(* Logix 5000 project; controller Final vendor 1 type 14 code 242 rev 32.11; software revision 32.00 *)

TASK MainTask (continuous, watchdog 500 ms) : MainProgram
TASK SafetyTask (periodic, rate 20 ms, priority 10, watchdog 20 ms, safety) : SafetyProgram

MODULES
   Local : vendor 1 type 14 code 242 (5069 0, rev 32.11)
      IO_002 : 5069-IF8 (5069 2, rev 2.1, StandardDataDriven RPI 100 ms)
      IO_001 : 5069-IF8 (5069 1, rev 2.1, StandardDataDriven RPI 100 ms)
      IO_003 : 5069-IF8 (5069 3, rev 2.1, StandardDataDriven RPI 100 ms)
      IO_006 : vendor 1 type 7 code 394 (5069 6, rev 2.1, StandardDataDriven RPI 5 ms)
      IO_004 : vendor 1 type 7 code 395 (5069 4, rev 2.1, StandardDataDriven RPI 5 ms)
      IO_005 : vendor 1 type 7 code 395 (5069 5, rev 2.1, StandardDataDriven RPI 5 ms)
      IO_007 : vendor 1 type 109 code 90 (5069 7, rev 3.1, StandardDataDriven RPI 80 ms)
      EN_001 : 1734-AENTR (Ethernet 107.0.114.14, rev 5.1, Output RPI 20 ms)
         IO_008 : vendor 1 type 35 code 15 (PointIO 1, rev 2.1, Input RPI 10 ms, Output RPI 20 ms)
         IO_009 : vendor 1 type 35 code 16 (PointIO 2, rev 2.1, Input RPI 10 ms, Output RPI 20 ms)
END_MODULES

TYPE SensorType :   // To monitor the sensor readings, we use this data type
STRUCT
   CurrentValue : DINT;
   PreviousValue0 : DINT;
   PreviousValue1 : DINT;
   PreviousValue2 : DINT;
   PreviousValue3 : DINT;
   PreviousValue4 : DINT;
   PreviousValue5 : DINT;
   PreviousValue6 : DINT;
   PreviousValue7 : DINT;
   PreviousValue8 : DINT;
   PreviousValue9 : DINT;
   Mean10 : DINT;
   StanDev : DINT;
   State : DINT;
   Count : DINT;
   MeanStart : BOOL;
END_STRUCT
END_TYPE

VAR_GLOBAL   (* controller tags *)
   ACC_TIMER : DINT;
   AT : BOOL;
   B_NomCount : DINT;
   B_Pres0 : SensorType;   // Holds all values related to Brakes Pressure Sensor #0
   B_Pres1 : SensorType;   // Holds all values related to Brakes Pressure Sensor #1
   B_Pres2 : SensorType;   // Holds all values related to Brakes Pressure Sensor #2
   B_Pres3 : SensorType;   // Holds all values related to Brakes Pressure Sensor #3
   B_Pres4 : SensorType;   // Holds all values related to Brakes Pressure Sensor #4
   B_Pres5 : SensorType;   // Holds all values related to Brakes Pressure Sensor #5
   B_Pres6 : SensorType;   // Holds all values related to Brakes Pressure Sensor #6
   B_Pres7 : SensorType;   // Holds all values related to Brakes Pressure Sensor #7
   B_Pres8 : SensorType;   // Holds all values related to Brakes Pressure Sensor #8
   B_Pres9 : SensorType;   // Holds all values related to Brakes Pressure Sensor #9
   B_Tem0 : SensorType;   // Holds all values related to Brakes Temperature Sensor #0
   B_Tem1 : SensorType;   // Holds all values related to Brakes Temperature Sensor #1
   BAT_FLAG : DINT;
   BATTERY_CURRENT : DINT;
   BATTERY_TEMP : DINT;
   BATTERY_VOLTAGE : DINT;
   BRAKE_FLAG : DINT;
   BRAKE_SUBSTATE1 : DINT;
   BRAKE_SUBSTATE2 : DINT;
   C_Las0 : SensorType;   // Holds all values related to Controls Laser Sensor #0
   C_Las1 : SensorType;   // Holds all values related to Controls Laser Sensor #1
   CA : BOOL;
   CC : BOOL;
   CD1 : BOOL;
   CD2 : BOOL;
   CD3 : BOOL;
   COAST_TIMER : DINT;
   COAST_TONR : DINT;
   COMMAND : DINT;
   COMN_FLAG : DINT;
   CP1 : BOOL;
   CP2 : BOOL;
   CPX : BOOL;
   CT : BOOL;
   CurrentState : DINT;
   Initialized : DINT;
   P_NomCount : DINT;
   P_Pres0 : SensorType;   // Holds all values related to Pressure Pressure Sensor #0
   P_Pres1 : SensorType;   // Holds all values related to Pressure Pressure Sensor #1
   P_Pres2 : SensorType;   // Holds all values related to Pressure Pressure Sensor #2
   P_Pres3 : SensorType;
   P_Pres4 : SensorType;
   P_Tem0 : SensorType;   // Holds all values related to Pressure Temperature Sensor #0
   P_Tem1 : SensorType;   // Holds all values related to Pressure Temperature Sensor #1
   P_Tem2 : SensorType;
   P_Tem3 : SensorType;
   P_Tem4 : SensorType;
   POD_ACCELERATION : DINT;
   POD_DISTANCE : DINT;
   POD_TIME : DINT[2];
   POD_VELOCITY : DINT;
   PREV_ACCELERATION : DINT;
   PREV_DISTANCE : DINT;
   PREV_TIME : DINT[2];
   PREV_VELOCITY : DINT;
   PROP_FLAG : DINT;
   PROP_STATE : DINT;
   PROP_TNK_PRES : DINT;
   READY : BOOL;
   STATE : DINT;
   STRIPE_COUNT : DINT;
   SYSTEM_FAIL : DINT;
END_VAR

PROGRAM MainProgram   (* main routine MainRoutine *)
VAR
   ACC_TIMER : FBD_TIMER;
   COAST_TIMER : FBD_TIMER;
   SIMULATOR : FBD_TIMER;
END_VAR

ROUTINE A01_Initialize   (* structured text *)
// Initializes the values of all tags
   JSR(Initial_B_Pres0);
   JSR(Initial_B_Pres1);
   JSR(Initial_B_Pres2);
   JSR(Initial_B_Pres3);
   JSR(Initial_B_Pres4);
   JSR(Initial_B_Pres5);
   JSR(Initial_B_Pres6);
   JSR(Initial_B_Pres7);
   JSR(Initial_B_Pres8);
   JSR(Initial_B_Pres9);
   JSR(Initial_B_Tem0);
   JSR(Initial_B_Tem1);
   Local:5:O.Pt00.Data := 1;
   Local:5:O.Pt01.Data := 1;
   Local:5:O.Pt02.Data := 1;
   Local:5:O.Pt03.Data := 1;
   B_NomCount := 24; //Brakes Initialized
   JSR(Initial_C_Las0);
   JSR(Initial_C_Las1); //Controls Initialized
   JSR(Initial_P_Pres0);
   JSR(Initial_P_Pres1);
   JSR(Initial_P_Pres2);
   JSR(Initial_P_Pres3);
   JSR(Initial_P_Pres4);
   JSR(Initial_P_Tem0);
   JSR(Initial_P_Tem1);
   JSR(Initial_P_Tem2);
   JSR(Initial_P_Tem3);
   JSR(Initial_P_Tem4);
   Local:4:O.Pt00.Data := 1;
   Local:4:O.Pt01.Data := 0;
   Local:4:O.Pt02.Data := 0;
   Local:4:O.Pt03.Data := 1;
   P_NomCount := 20; //Propulsion Initialized
   BATTERY_CURRENT := 0;
   BATTERY_TEMP := 0;
   BATTERY_VOLTAGE := 0; //Power Initialized
   STRIPE_COUNT := 0;
   POD_DISTANCE := 0;
   POD_VELOCITY := 0;
   POD_ACCELERATION := 0;
   PREV_DISTANCE := 0;
   PREV_VELOCITY := 0;
   PREV_ACCELERATION := 0;
   READY := 0;
   //COAST_TIMER := 0;
   PROP_TNK_PRES := 0;
   PROP_STATE := 0;
   BRAKE_SUBSTATE1 := 0;
   BRAKE_SUBSTATE2 := 0;
   PROP_FLAG := 0;
   BRAKE_FLAG := 0;
   COMN_FLAG := 0;
   BAT_FLAG := 0;
   SYSTEM_FAIL := 0;
   STATE := 1;
   Initialized := 5380; //All Initialized
   //low-speed drive parameters missing
END_ROUTINE

ROUTINE A02_Update   (* structured text *)
// Updates all sensor value tags
   JSR(Update_B_Pres0);
   JSR(Update_B_Pres1);
   JSR(Update_B_Pres2);
   JSR(Update_B_Pres3);
   JSR(Update_B_Pres4);
   JSR(Update_B_Pres5);
   JSR(Update_B_Pres6);
   JSR(Update_B_Pres7);
   JSR(Update_B_Pres8);
   JSR(Update_B_Pres9);
   JSR(Update_B_Tem0);
   JSR(Update_B_Tem1); //Brakes Updated
   JSR(Update_C_Las0);
   JSR(Update_C_Las1); //Controls Updated
   JSR(Update_P_Pres0);
   JSR(Update_P_Pres1);
   JSR(Update_P_Pres2);
   JSR(Update_P_Pres3);
   JSR(Update_P_Pres4);
   JSR(Update_P_Tem0);
   JSR(Update_P_Tem1);
   JSR(Update_P_Tem2);
   JSR(Update_P_Tem3);
   JSR(Update_P_Tem4); //Propulsion Updated
   JSR(Update_Bat_Current);
   JSR(Update_Bat_Temp);
   JSR(Update_Bat_Voltage); //Power Updated
   JSR(Rx_Command);
   //limit switches
   //low-speed drive parameters
END_ROUTINE

ROUTINE A03_Process   (* structured text *)
// Processes input data
   //high speed counter interface
   STRIPE_COUNT := (C_Las0.CurrentValue + C_Las1.CurrentValue)/2; //2 can be substituted with nominal count of laser sensors
   
   PREV_DISTANCE := POD_DISTANCE;
   POD_DISTANCE := STRIPE_COUNT*3048; //units cm
   
   PREV_TIME[0] := POD_TIME[0];
   GSV(WallClockTime,,CurrentValue,POD_TIME[0]); //units microseconds
   
   PREV_VELOCITY := POD_VELOCITY;
   POD_VELOCITY := (POD_DISTANCE - PREV_DISTANCE)/(100000*(POD_TIME[0] - PREV_TIME[0])); //units cm/s
   
   PREV_ACCELERATION := POD_ACCELERATION;
   POD_ACCELERATION := (POD_VELOCITY - PREV_VELOCITY)/(POD_TIME[0] - PREV_TIME[0]); //units cm/s2
   
   //Process Data part 2
END_ROUTINE

ROUTINE A04_State   (* structured text *)
// Updates the state of the pod
   JSR(Check_Distance_1); //Checks if POD_DISTANCE >= 3000 cm
   JSR(Check_Distance_2); //Checks if POD_DISTANCE >= 80000 cm
   JSR(Check_Distance_3); //Checks if POD_DISTANCE >= 125000 cm
   JSR(Check_TankPres_1); //Checks if PROP_TNK_PRES >= 200 PSI
   JSR(Check_TankPres_2); //Checks if PROP_TNK_PRES <= 100 PSI
   JSR(Check_TankPres_X); //Checks if ACT_TNK_PRES == ??
   JSR(Check_PodAcc_1); //Checks if POD_ACCELERATION <= 0 cm/s2
   JSR(Check_AccTimer); // Checks if ACC_TIMER >= 7.7 sec
   JSR(Check_CoastTimer); //Checks if COAST_TIMER >= 10 sec
END_ROUTINE

ROUTINE A05_Actions   (* structured text *)
// Performs the state actions of the pod
   case STATE of
   	1: JSR(B01_Idle);
   	2: JSR(B02_SystemCheck);
   	3: JSR(B03_Armed);
   	4: JSR(B04_Acceleration);
   	5: JSR(B05_Coast);
   	6: JSR(B06_Brake);
   	7: JSR(B07_Stop);
   	8: JSR(B08_Crawl);
   	9: JSR(B09_End);
   	10: JSR(B10_EmergencyShutdown);
   end_case;
END_ROUTINE

ROUTINE A06_Relay   (* structured text *)
// Relays pod data to monitoring station
   //communication
END_ROUTINE

ROUTINE B01_Idle   (* structured text *)
   if COMMAND = 2 then
   	STATE := 2; //System Check
   end_if;
   
   if COMMAND = 9 then
   	STATE := 9; //End
   end_if;
   
   if COMMAND = 10 then
   	STATE := 10; //Emergency Shutdown
   end_if;
END_ROUTINE

ROUTINE B02_SystemCheck   (* structured text *)
   JSR(NomCheck_B1);
   JSR(NomCheck_P1);
   
   if B_NomCount <> 24 then
   	JSR(FaultTest_B);
   end_if;
   
   if P_NomCount <> 24 then
   	JSR(FaultTest_P);
   end_if;
   
   if COMMAND = 3 then
   	STATE := 3; //Armed
   end_if;
   
   if COMMAND = 1 then
   	STATE := 1; //Idle
   end_if;
   
   if COMMAND = 10 then
   	STATE := 10; //Emergency Shutdown
   end_if;
END_ROUTINE

ROUTINE B03_Armed   (* structured text *)
   if COMMAND = 4 then
   	STATE := 4; //Acceleration
   end_if;
   
   if COMMAND = 8 then
   	STATE := 8; //Crawl
   end_if;
   
   if COMMAND = 10 then
   	STATE := 10; //Emergency Shutdown
   end_if;
END_ROUTINE

ROUTINE B04_Acceleration   (* structured text *)
   ACC_TIMER.PRE := 10000;
   ACC_TIMER.TimerEnable := 1;
   ACC_TIMER.Reset := 0;
   TONR(ACC_TIMER);
   
   //EN_001:2:O.Pt01Data := 1;
   //EN_001:2:O.Pt02Data := 1;
   //EN_001:2:O.Pt00Data := 1; //Slow crawl
   
   if CD1 then //POD_DISTANCE >= 3000 cm?
   	//EN_001:2:O.Pt01Data := 0;
   	//EN_001:2:O.Pt02Data := 0;
   	//EN_001:2:O.Pt00Data := 0; //End crawl
   	READY := 1;
   end_if;
   //Timer to ready
   if READY then
   	Local:4:O.Pt01.Data := 1;
   	Local:4:O.Pt02.Data := 1; //Activate Propulsion
   end_if;
   
   if CPX then //TA-5 > 900 PSI?
   	Local:4:O.Pt00.Data := 0; //Special condition
   end_if;
   
   if CP1 AND CA then //PROP_TNK_PRES <= 200 PSI?
   	STATE := 5; //Coast
   end_if;
END_ROUTINE

ROUTINE B05_Coast   (* structured text *)
   COAST_TIMER.PRE := 7700;
   COAST_TIMER.TimerEnable := 1;
   COAST_TIMER.Reset := 0;
   TONR(COAST_TIMER); //Coast timer initialized
   
   Local:4:O.Pt01.Data := 0;
   Local:4:O.Pt02.Data := 0; //Propulsion disengaged
   
   if CP2 then
   	Local:4:O.Pt03.Data := 0; //Relief pressure valve open
   end_if;
   
   if CD2 OR CT OR (COMMAND = 7) then
   	STATE := 6; //Brake
   end_if;
   
   if COMMAND = 10 then
   	STATE := 10; //Emergency Shutdown
   end_if;
END_ROUTINE

ROUTINE B06_Brake   (* structured text *)
   Local:4:O.Pt03.Data := 1; //Relief pressure valve closed
   Local:5:O.Pt00.Data := 0;
   Local:5:O.Pt01.Data := 0;
   Local:5:O.Pt02.Data := 0;
   Local:5:O.Pt03.Data := 0; //Brakes engaged
   
   if POD_VELOCITY = 0 then
   	STATE := 7; //Stop
   end_if;
   
   if CA then
   	STATE := 10;
   end_if;
END_ROUTINE

ROUTINE B07_Stop   (* structured text *)
   Local:5:O.Pt00.Data := 1;
   Local:5:O.Pt01.Data := 1;
   Local:5:O.Pt02.Data := 1;
   Local:5:O.Pt03.Data := 1; //Disengage Brakes
   
   if COMMAND = 8 then
   STATE := 8; //Crawl
   end_if;
   
   if COMMAND = 9 then
   STATE := 9; //End
   end_if;
   
   if COMMAND = 10 then
   	STATE := 10; //Emergency Shutdown
   end_if;
END_ROUTINE

ROUTINE B08_Crawl   (* structured text *)
   //EN_001:2:O.Pt01Data := 1; // D = 1 Forward, D = 0 Backward
   //EN_001:2:O.Pt02Data := 1; //
   //EN_001:2:O.Pt00Data := 1; // pulse F at 4333 Hz //Slow crawl
   
   if CD3 OR (COMMAND = 7) then
   	//EN_001:2:O.Pt01Data := 0;
   	//EN_001:2:O.Pt02Data := 0;
   	//EN_001:2:O.Pt00Data := 0; //End crawl
   	STATE := 6; //Stop
   end_if;
END_ROUTINE

ROUTINE B09_End   (* structured text *)
   //Do nothing
END_ROUTINE

ROUTINE B10_EmergencyShutdown   (* structured text *)
   // Relay system faliure
   if CA then
   	Local:4:O.Pt01.Data := 0;
   	Local:4:O.Pt02.Data := 0; //Propulsion tanks closed
   end_if;
   Local:5:O.Pt00.Data := 0;
   Local:5:O.Pt01.Data := 0;
   Local:5:O.Pt02.Data := 0;
   Local:5:O.Pt03.Data := 0; //Brakes activated
   
   if CP2 then
   	STATE := 7; //Stop
   else
   	Local:4:O.Pt03.Data := 0; //Relief pressure valve
   	STATE := 7; //Stop
   end_if;
END_ROUTINE

ROUTINE Check_AccTimer   (* structured text *)
   if ACC_TIMER.DN then
   	AT := 1;
   	end_if;
END_ROUTINE

ROUTINE Check_CoastTimer   (* structured text *)
   if COAST_TIMER.DN then
   	CT := 1;
   	end_if;
END_ROUTINE

ROUTINE Check_Distance_1   (* structured text *)
   if POD_DISTANCE >= 3000 then
   	CD1 := 1;
   end_if;
END_ROUTINE

ROUTINE Check_Distance_2   (* structured text *)
   if POD_DISTANCE >= 80000 then
   	CD2 := 1;
   end_if;
END_ROUTINE

ROUTINE Check_Distance_3   (* structured text *)
   if POD_DISTANCE >= 125000 then
   	CD3 := 1;
   end_if;
END_ROUTINE

ROUTINE Check_LSDTimer   (* structured text *)
   
END_ROUTINE

ROUTINE Check_PodAcc_1   (* structured text *)
   if POD_ACCELERATION <= 0 then
   	CA := 1;
   end_if;
END_ROUTINE

ROUTINE Check_TankPres_1   (* structured text *)
   if (P_Pres1.CurrentValue + P_Pres2.CurrentValue + P_Pres3.CurrentValue + P_Pres4.CurrentValue) <= 200 then
   	CP1 := 1;
   end_if;
END_ROUTINE

ROUTINE Check_TankPres_2   (* structured text *)
   if (P_Pres1.CurrentValue + P_Pres2.CurrentValue + P_Pres3.CurrentValue + P_Pres4.CurrentValue) = 0 then
   	CP2 := 1;
   end_if;
END_ROUTINE

ROUTINE Check_TankPres_X   (* structured text *)
   if P_Pres0.CurrentValue < 250 then
   	CPX := 1;
   end_if;
END_ROUTINE

ROUTINE FaultTest_B   (* structured text *)
   
END_ROUTINE

ROUTINE FaultTest_P   (* structured text *)
   
END_ROUTINE

ROUTINE Initial_B_Pres0   (* structured text *)
   B_Pres0.CurrentValue := 0;
   B_Pres0.PreviousValue0 := 0;
   B_Pres0.PreviousValue1 := 0;
   B_Pres0.PreviousValue2 := 0;
   B_Pres0.PreviousValue3 := 0;
   B_Pres0.PreviousValue4 := 0;
   B_Pres0.PreviousValue5 := 0;
   B_Pres0.PreviousValue6 := 0;
   B_Pres0.PreviousValue7 := 0;
   B_Pres0.PreviousValue8 := 0;
   B_Pres0.PreviousValue9 := 0;
   B_Pres0.Count := 0;
   B_Pres0.Mean10 := 0;
   B_Pres0.StanDev := 0;
   B_Pres0.State := 0;
   B_Pres0.MeanStart := 0;
END_ROUTINE

ROUTINE Initial_B_Pres1   (* structured text *)
   B_Pres1.CurrentValue := 0;
   B_Pres1.PreviousValue0 := 0;
   B_Pres1.PreviousValue1 := 0;
   B_Pres1.PreviousValue2 := 0;
   B_Pres1.PreviousValue3 := 0;
   B_Pres1.PreviousValue4 := 0;
   B_Pres1.PreviousValue5 := 0;
   B_Pres1.PreviousValue6 := 0;
   B_Pres1.PreviousValue7 := 0;
   B_Pres1.PreviousValue8 := 0;
   B_Pres1.PreviousValue9 := 0;
   B_Pres1.Count := 0;
   B_Pres1.Mean10 := 0;
   B_Pres1.StanDev := 0;
   B_Pres1.State := 0;
   B_Pres1.MeanStart := 0;
END_ROUTINE

ROUTINE Initial_B_Pres2   (* structured text *)
   B_Pres2.CurrentValue := 0;
   B_Pres2.PreviousValue0 := 0;
   B_Pres2.PreviousValue1 := 0;
   B_Pres2.PreviousValue2 := 0;
   B_Pres2.PreviousValue3 := 0;
   B_Pres2.PreviousValue4 := 0;
   B_Pres2.PreviousValue5 := 0;
   B_Pres2.PreviousValue6 := 0;
   B_Pres2.PreviousValue7 := 0;
   B_Pres2.PreviousValue8 := 0;
   B_Pres2.PreviousValue9 := 0;
   B_Pres2.Count := 0;
   B_Pres2.Mean10 := 0;
   B_Pres2.StanDev := 0;
   B_Pres2.State := 0;
   B_Pres2.MeanStart := 0;
END_ROUTINE

ROUTINE Initial_B_Pres3   (* structured text *)
   B_Pres3.CurrentValue := 0;
   B_Pres3.PreviousValue0 := 0;
   B_Pres3.PreviousValue1 := 0;
   B_Pres3.PreviousValue2 := 0;
   B_Pres3.PreviousValue3 := 0;
   B_Pres3.PreviousValue4 := 0;
   B_Pres3.PreviousValue5 := 0;
   B_Pres3.PreviousValue6 := 0;
   B_Pres3.PreviousValue7 := 0;
   B_Pres3.PreviousValue8 := 0;
   B_Pres3.PreviousValue9 := 0;
   B_Pres3.Count := 0;
   B_Pres3.Mean10 := 0;
   B_Pres3.StanDev := 0;
   B_Pres3.State := 0;
   B_Pres3.MeanStart := 0;
END_ROUTINE

ROUTINE Initial_B_Pres4   (* structured text *)
   B_Pres4.CurrentValue := 0;
   B_Pres4.PreviousValue0 := 0;
   B_Pres4.PreviousValue1 := 0;
   B_Pres4.PreviousValue2 := 0;
   B_Pres4.PreviousValue3 := 0;
   B_Pres4.PreviousValue4 := 0;
   B_Pres4.PreviousValue5 := 0;
   B_Pres4.PreviousValue6 := 0;
   B_Pres4.PreviousValue7 := 0;
   B_Pres4.PreviousValue8 := 0;
   B_Pres4.PreviousValue9 := 0;
   B_Pres4.Count := 0;
   B_Pres4.Mean10 := 0;
   B_Pres4.StanDev := 0;
   B_Pres4.State := 0;
   B_Pres4.MeanStart := 0;
END_ROUTINE

ROUTINE Initial_B_Pres5   (* structured text *)
   B_Pres5.CurrentValue := 0;
   B_Pres5.PreviousValue0 := 0;
   B_Pres5.PreviousValue1 := 0;
   B_Pres5.PreviousValue2 := 0;
   B_Pres5.PreviousValue3 := 0;
   B_Pres5.PreviousValue4 := 0;
   B_Pres5.PreviousValue5 := 0;
   B_Pres5.PreviousValue6 := 0;
   B_Pres5.PreviousValue7 := 0;
   B_Pres5.PreviousValue8 := 0;
   B_Pres5.PreviousValue9 := 0;
   B_Pres5.Count := 0;
   B_Pres5.Mean10 := 0;
   B_Pres5.StanDev := 0;
   B_Pres5.State := 0;
   B_Pres5.MeanStart := 0;
END_ROUTINE

ROUTINE Initial_B_Pres6   (* structured text *)
   B_Pres6.CurrentValue := 0;
   B_Pres6.PreviousValue0 := 0;
   B_Pres6.PreviousValue1 := 0;
   B_Pres6.PreviousValue2 := 0;
   B_Pres6.PreviousValue3 := 0;
   B_Pres6.PreviousValue4 := 0;
   B_Pres6.PreviousValue5 := 0;
   B_Pres6.PreviousValue6 := 0;
   B_Pres6.PreviousValue7 := 0;
   B_Pres6.PreviousValue8 := 0;
   B_Pres6.PreviousValue9 := 0;
   B_Pres6.Count := 0;
   B_Pres6.Mean10 := 0;
   B_Pres6.StanDev := 0;
   B_Pres6.State := 0;
   B_Pres6.MeanStart := 0;
END_ROUTINE

ROUTINE Initial_B_Pres7   (* structured text *)
   B_Pres7.CurrentValue := 0;
   B_Pres7.PreviousValue0 := 0;
   B_Pres7.PreviousValue1 := 0;
   B_Pres7.PreviousValue2 := 0;
   B_Pres7.PreviousValue3 := 0;
   B_Pres7.PreviousValue4 := 0;
   B_Pres7.PreviousValue5 := 0;
   B_Pres7.PreviousValue6 := 0;
   B_Pres7.PreviousValue7 := 0;
   B_Pres7.PreviousValue8 := 0;
   B_Pres7.PreviousValue9 := 0;
   B_Pres7.Count := 0;
   B_Pres7.Mean10 := 0;
   B_Pres7.StanDev := 0;
   B_Pres7.State := 0;
   B_Pres7.MeanStart := 0;
END_ROUTINE

ROUTINE Initial_B_Pres8   (* structured text *)
   B_Pres8.CurrentValue := 0;
   B_Pres8.PreviousValue0 := 0;
   B_Pres8.PreviousValue1 := 0;
   B_Pres8.PreviousValue2 := 0;
   B_Pres8.PreviousValue3 := 0;
   B_Pres8.PreviousValue4 := 0;
   B_Pres8.PreviousValue5 := 0;
   B_Pres8.PreviousValue6 := 0;
   B_Pres8.PreviousValue7 := 0;
   B_Pres8.PreviousValue8 := 0;
   B_Pres8.PreviousValue9 := 0;
   B_Pres8.Count := 0;
   B_Pres8.Mean10 := 0;
   B_Pres8.StanDev := 0;
   B_Pres8.State := 0;
   B_Pres8.MeanStart := 0;
END_ROUTINE

ROUTINE Initial_B_Pres9   (* structured text *)
   B_Pres9.CurrentValue := 0;
   B_Pres9.PreviousValue0 := 0;
   B_Pres9.PreviousValue1 := 0;
   B_Pres9.PreviousValue2 := 0;
   B_Pres9.PreviousValue3 := 0;
   B_Pres9.PreviousValue4 := 0;
   B_Pres9.PreviousValue5 := 0;
   B_Pres9.PreviousValue6 := 0;
   B_Pres9.PreviousValue7 := 0;
   B_Pres9.PreviousValue8 := 0;
   B_Pres9.PreviousValue9 := 0;
   B_Pres9.Count := 0;
   B_Pres9.Mean10 := 0;
   B_Pres9.StanDev := 0;
   B_Pres9.State := 0;
   B_Pres9.MeanStart := 0;
END_ROUTINE

ROUTINE Initial_B_Tem0   (* structured text *)
   B_Tem0.CurrentValue := 0;
   B_Tem0.PreviousValue0 := 0;
   B_Tem0.PreviousValue1 := 0;
   B_Tem0.PreviousValue2 := 0;
   B_Tem0.PreviousValue3 := 0;
   B_Tem0.PreviousValue4 := 0;
   B_Tem0.PreviousValue5 := 0;
   B_Tem0.PreviousValue6 := 0;
   B_Tem0.PreviousValue7 := 0;
   B_Tem0.PreviousValue8 := 0;
   B_Tem0.PreviousValue9 := 0;
   B_Tem0.Count := 0;
   B_Tem0.Mean10 := 0;
   B_Tem0.StanDev := 0;
   B_Tem0.State := 0;
   B_Tem0.MeanStart := 0;
END_ROUTINE

ROUTINE Initial_B_Tem1   (* structured text *)
   B_Tem1.CurrentValue := 0;
   B_Tem1.PreviousValue0 := 0;
   B_Tem1.PreviousValue1 := 0;
   B_Tem1.PreviousValue2 := 0;
   B_Tem1.PreviousValue3 := 0;
   B_Tem1.PreviousValue4 := 0;
   B_Tem1.PreviousValue5 := 0;
   B_Tem1.PreviousValue6 := 0;
   B_Tem1.PreviousValue7 := 0;
   B_Tem1.PreviousValue8 := 0;
   B_Tem1.PreviousValue9 := 0;
   B_Tem1.Count := 0;
   B_Tem1.Mean10 := 0;
   B_Tem1.StanDev := 0;
   B_Tem1.State := 0;
   B_Tem1.MeanStart := 0;
END_ROUTINE

ROUTINE Initial_C_Las0   (* structured text *)
   C_Las0.CurrentValue := 0;
   C_Las0.PreviousValue0 := 0;
   C_Las0.PreviousValue1 := 0;
   C_Las0.PreviousValue2 := 0;
   C_Las0.PreviousValue3 := 0;
   C_Las0.PreviousValue4 := 0;
   C_Las0.PreviousValue5 := 0;
   C_Las0.PreviousValue6 := 0;
   C_Las0.PreviousValue7 := 0;
   C_Las0.PreviousValue8 := 0;
   C_Las0.PreviousValue9 := 0;
   C_Las0.Count := 0;
   C_Las0.Mean10 := 0;
   C_Las0.StanDev := 0;
   C_Las0.State := 0;
   C_Las0.MeanStart := 0;
END_ROUTINE

ROUTINE Initial_C_Las1   (* structured text *)
   C_Las1.CurrentValue := 0;
   C_Las1.PreviousValue0 := 0;
   C_Las1.PreviousValue1 := 0;
   C_Las1.PreviousValue2 := 0;
   C_Las1.PreviousValue3 := 0;
   C_Las1.PreviousValue4 := 0;
   C_Las1.PreviousValue5 := 0;
   C_Las1.PreviousValue6 := 0;
   C_Las1.PreviousValue7 := 0;
   C_Las1.PreviousValue8 := 0;
   C_Las1.PreviousValue9 := 0;
   C_Las1.Count := 0;
   C_Las1.Mean10 := 0;
   C_Las1.StanDev := 0;
   C_Las1.State := 0;
   C_Las0.MeanStart := 0;
END_ROUTINE

ROUTINE Initial_P_Pres0   (* structured text *)
   P_Pres0.CurrentValue := 0;
   P_Pres0.PreviousValue0 := 0;
   P_Pres0.PreviousValue1 := 0;
   P_Pres0.PreviousValue2 := 0;
   P_Pres0.PreviousValue3 := 0;
   P_Pres0.PreviousValue4 := 0;
   P_Pres0.PreviousValue5 := 0;
   P_Pres0.PreviousValue6 := 0;
   P_Pres0.PreviousValue7 := 0;
   P_Pres0.PreviousValue8 := 0;
   P_Pres0.PreviousValue9 := 0;
   P_Pres0.Count := 0;
   P_Pres0.Mean10 := 0;
   P_Pres0.StanDev := 0;
   P_Pres0.State := 0;
   P_Pres0.MeanStart := 0;
END_ROUTINE

ROUTINE Initial_P_Pres1   (* structured text *)
   P_Pres1.CurrentValue := 0;
   P_Pres1.PreviousValue0 := 0;
   P_Pres1.PreviousValue1 := 0;
   P_Pres1.PreviousValue2 := 0;
   P_Pres1.PreviousValue3 := 0;
   P_Pres1.PreviousValue4 := 0;
   P_Pres1.PreviousValue5 := 0;
   P_Pres1.PreviousValue6 := 0;
   P_Pres1.PreviousValue7 := 0;
   P_Pres1.PreviousValue8 := 0;
   P_Pres1.PreviousValue9 := 0;
   P_Pres1.Count := 0;
   P_Pres1.Mean10 := 0;
   P_Pres1.StanDev := 0;
   P_Pres1.State := 0;
   P_Pres1.MeanStart := 0;
END_ROUTINE

ROUTINE Initial_P_Pres2   (* structured text *)
   P_Pres2.CurrentValue := 0;
   P_Pres2.PreviousValue0 := 0;
   P_Pres2.PreviousValue1 := 0;
   P_Pres2.PreviousValue2 := 0;
   P_Pres2.PreviousValue3 := 0;
   P_Pres2.PreviousValue4 := 0;
   P_Pres2.PreviousValue5 := 0;
   P_Pres2.PreviousValue6 := 0;
   P_Pres2.PreviousValue7 := 0;
   P_Pres2.PreviousValue8 := 0;
   P_Pres2.PreviousValue9 := 0;
   P_Pres2.Count := 0;
   P_Pres2.Mean10 := 0;
   P_Pres2.StanDev := 0;
   P_Pres2.State := 0;
   P_Pres2.MeanStart := 0;
END_ROUTINE

ROUTINE Initial_P_Pres3   (* structured text *)
   P_Pres3.CurrentValue := 0;
   P_Pres3.PreviousValue0 := 0;
   P_Pres3.PreviousValue1 := 0;
   P_Pres3.PreviousValue2 := 0;
   P_Pres3.PreviousValue3 := 0;
   P_Pres3.PreviousValue4 := 0;
   P_Pres3.PreviousValue5 := 0;
   P_Pres3.PreviousValue6 := 0;
   P_Pres3.PreviousValue7 := 0;
   P_Pres3.PreviousValue8 := 0;
   P_Pres3.PreviousValue9 := 0;
   P_Pres3.Count := 0;
   P_Pres3.Mean10 := 0;
   P_Pres3.StanDev := 0;
   P_Pres3.State := 0;
   P_Pres3.MeanStart := 0;
END_ROUTINE

ROUTINE Initial_P_Pres4   (* structured text *)
   P_Pres4.CurrentValue := 0;
   P_Pres4.PreviousValue0 := 0;
   P_Pres4.PreviousValue1 := 0;
   P_Pres4.PreviousValue2 := 0;
   P_Pres4.PreviousValue3 := 0;
   P_Pres4.PreviousValue4 := 0;
   P_Pres4.PreviousValue5 := 0;
   P_Pres4.PreviousValue6 := 0;
   P_Pres4.PreviousValue7 := 0;
   P_Pres4.PreviousValue8 := 0;
   P_Pres4.PreviousValue9 := 0;
   P_Pres4.Count := 0;
   P_Pres4.Mean10 := 0;
   P_Pres4.StanDev := 0;
   P_Pres4.State := 0;
   P_Pres4.MeanStart := 0;
END_ROUTINE

ROUTINE Initial_P_Tem0   (* structured text *)
   P_Tem0.CurrentValue := 0;
   P_Tem0.PreviousValue0 := 0;
   P_Tem0.PreviousValue1 := 0;
   P_Tem0.PreviousValue2 := 0;
   P_Tem0.PreviousValue3 := 0;
   P_Tem0.PreviousValue4 := 0;
   P_Tem0.PreviousValue5 := 0;
   P_Tem0.PreviousValue6 := 0;
   P_Tem0.PreviousValue7 := 0;
   P_Tem0.PreviousValue8 := 0;
   P_Tem0.PreviousValue9 := 0;
   P_Tem0.Count := 0;
   P_Tem0.Mean10 := 0;
   P_Tem0.StanDev := 0;
   P_Tem0.State := 0;
   P_Tem0.MeanStart := 0;
END_ROUTINE

ROUTINE Initial_P_Tem1   (* structured text *)
   P_Tem1.CurrentValue := 0;
   P_Tem1.PreviousValue0 := 0;
   P_Tem1.PreviousValue1 := 0;
   P_Tem1.PreviousValue2 := 0;
   P_Tem1.PreviousValue3 := 0;
   P_Tem1.PreviousValue4 := 0;
   P_Tem1.PreviousValue5 := 0;
   P_Tem1.PreviousValue6 := 0;
   P_Tem1.PreviousValue7 := 0;
   P_Tem1.PreviousValue8 := 0;
   P_Tem1.PreviousValue9 := 0;
   P_Tem1.Count := 0;
   P_Tem1.Mean10 := 0;
   P_Tem1.StanDev := 0;
   P_Tem1.State := 0;
   P_Tem1.MeanStart := 0;
END_ROUTINE

ROUTINE Initial_P_Tem2   (* structured text *)
   P_Tem2.CurrentValue := 0;
   P_Tem2.PreviousValue0 := 0;
   P_Tem2.PreviousValue1 := 0;
   P_Tem2.PreviousValue2 := 0;
   P_Tem2.PreviousValue3 := 0;
   P_Tem2.PreviousValue4 := 0;
   P_Tem2.PreviousValue5 := 0;
   P_Tem2.PreviousValue6 := 0;
   P_Tem2.PreviousValue7 := 0;
   P_Tem2.PreviousValue8 := 0;
   P_Tem2.PreviousValue9 := 0;
   P_Tem2.Count := 0;
   P_Tem2.Mean10 := 0;
   P_Tem2.StanDev := 0;
   P_Tem2.State := 0;
   P_Tem2.MeanStart := 0;
END_ROUTINE

ROUTINE Initial_P_Tem3   (* structured text *)
   P_Tem3.CurrentValue := 0;
   P_Tem3.PreviousValue0 := 0;
   P_Tem3.PreviousValue1 := 0;
   P_Tem3.PreviousValue2 := 0;
   P_Tem3.PreviousValue3 := 0;
   P_Tem3.PreviousValue4 := 0;
   P_Tem3.PreviousValue5 := 0;
   P_Tem3.PreviousValue6 := 0;
   P_Tem3.PreviousValue7 := 0;
   P_Tem3.PreviousValue8 := 0;
   P_Tem3.PreviousValue9 := 0;
   P_Tem3.Count := 0;
   P_Tem3.Mean10 := 0;
   P_Tem3.StanDev := 0;
   P_Tem3.State := 0;
   P_Tem3.MeanStart := 0;
END_ROUTINE

ROUTINE Initial_P_Tem4   (* structured text *)
   P_Tem4.CurrentValue := 0;
   P_Tem4.PreviousValue0 := 0;
   P_Tem4.PreviousValue1 := 0;
   P_Tem4.PreviousValue2 := 0;
   P_Tem4.PreviousValue3 := 0;
   P_Tem4.PreviousValue4 := 0;
   P_Tem4.PreviousValue5 := 0;
   P_Tem4.PreviousValue6 := 0;
   P_Tem4.PreviousValue7 := 0;
   P_Tem4.PreviousValue8 := 0;
   P_Tem4.PreviousValue9 := 0;
   P_Tem4.Count := 0;
   P_Tem4.Mean10 := 0;
   P_Tem4.StanDev := 0;
   P_Tem4.State := 0;
   P_Tem4.MeanStart := 0;
END_ROUTINE

ROUTINE MainRoutine   (* structured text *)
// The main routine
   if Initialized = 5380 then //Initialized?
   JSR(A02_Update);
   JSR(A03_Process);
   JSR(A04_State);
   JSR(A05_Actions);
   JSR(A06_Relay);
   else
   JSR(A01_Initialize);
   end_if;
END_ROUTINE

ROUTINE NomCheck_B1   (* structured text *)
   if (B_Pres0.CurrentValue > 105) OR (B_Pres0.CurrentValue < 95) then
   		B_Pres0.State := 2;
   else B_Pres0.State := 0;
   end_if;
   if (B_Pres1.CurrentValue > 105) OR (B_Pres1.CurrentValue < 95) then
   		B_Pres1.State := 2;
   else B_Pres1.State := 0;
   end_if;
   if (B_Pres5.CurrentValue > 105) OR (B_Pres5.CurrentValue < 95) then
   		B_Pres5.State := 2;
   else B_Pres5.State := 0;
   end_if;
   if (B_Pres6.CurrentValue > 105) OR (B_Pres6.CurrentValue < 95) then
   		B_Pres6.State := 2;
   else B_Pres6.State := 0;
   end_if;
   if (B_Pres2.CurrentValue > 16) OR (B_Pres2.CurrentValue < 12) then
   		B_Pres2.State := 2;
   else B_Pres2.State := 0;
   end_if;
   if (B_Pres3.CurrentValue > 16) OR (B_Pres3.CurrentValue < 12) then
   		B_Pres3.State := 2;
   else B_Pres3.State := 0;
   end_if;
   if (B_Pres7.CurrentValue > 16) OR (B_Pres7.CurrentValue < 12) then
   		B_Pres7.State := 2;
   else B_Pres7.State := 0;
   end_if;
   if (B_Pres8.CurrentValue > 16) OR (B_Pres8.CurrentValue < 12) then
   		B_Pres8.State := 2;
   else B_Pres8.State := 0;
   end_if;
   if (B_Pres4.CurrentValue > 170) OR (B_Pres4.CurrentValue < 150) then
   		B_Pres4.State := 2;
   else B_Pres4.State := 0;
   end_if;
   if (B_Pres9.CurrentValue > 170) OR (B_Pres9.CurrentValue < 150) then
   		B_Pres9.State := 2;
   else B_Pres9.State := 0;
   end_if;
   if (B_Tem0.CurrentValue > 30) OR (B_Tem0.CurrentValue < 20) then
   		B_Tem0.State := 2;
   else B_Tem0.State := 0;
   end_if;
   if (B_Tem1.CurrentValue > 30) OR (B_Tem1.CurrentValue < 20) then
   		B_Tem1.State := 2;
   else B_Tem1.State := 0;
   end_if;
   B_NomCount := 24 - (B_Pres0.State + B_Pres1.State + B_Pres2.State + B_Pres3.State + B_Pres4.State + B_Pres5.State + B_Pres6.State + B_Pres7.State + B_Pres8.State + B_Pres9.State + B_Tem0.State + B_Tem1.State);
END_ROUTINE

ROUTINE NomCheck_P1   (* structured text *)
   if P_Pres0.CurrentValue > 250 then
   	P_Pres0.State := 2;
   elsif P_Pres0.CurrentValue < 200 then
   	P_Pres0.State := 1;
   else P_Pres0.State := 0;
   end_if;
   if P_Pres1.CurrentValue > 3500 then
   	P_Pres1.State := 2;
   elsif P_Pres1.CurrentValue < 3000 then
   	P_Pres1.State := 1;
   else P_Pres1.State := 0;
   end_if;
   if P_Pres2.CurrentValue > 3500 then
   	P_Pres2.State := 2;
   elsif P_Pres2.CurrentValue < 3000 then
   	P_Pres2.State := 1;
   else P_Pres2.State := 0;
   end_if;
   if P_Pres3.CurrentValue > 3500 then
   	P_Pres3.State := 2;
   elsif P_Pres3.CurrentValue < 3000 then
   	P_Pres3.State := 1;
   else P_Pres3.State := 0;
   end_if;
   if P_Pres4.CurrentValue > 3500 then
   	P_Pres4.State := 2;
   elsif P_Pres4.CurrentValue < 3000 then
   	P_Pres4.State := 1;
   else P_Pres4.State := 0;
   end_if;
   if (P_Tem0.CurrentValue > 30) OR (P_Tem0.CurrentValue < 20) then
   		P_Tem0.State := 2;
   else P_Tem0.State := 0;
   end_if;
   if (P_Tem1.CurrentValue > 30) OR (P_Tem1.CurrentValue < 20) then
   		P_Tem1.State := 2;
   else P_Tem1.State := 0;
   end_if;
   if (P_Tem2.CurrentValue > 30) OR (P_Tem2.CurrentValue < 20) then
   		P_Tem2.State := 2;
   else P_Tem2.State := 0;
   end_if;
   if (P_Tem3.CurrentValue > 30) OR (P_Tem3.CurrentValue < 20) then
   		P_Tem3.State := 2;
   else P_Tem3.State := 0;
   end_if;
   if (P_Tem4.CurrentValue > 30) OR (P_Tem4.CurrentValue < 20) then
   		P_Tem4.State := 2;
   else P_Tem4.State := 0;
   end_if;
   P_NomCount := 20 - (P_Pres0.State + P_Pres1.State + P_Pres2.State + P_Pres3.State + P_Pres4.State + P_Tem0.State + P_Tem1.State + P_Tem2.State + P_Tem3.State + P_Tem4.State);
END_ROUTINE

ROUTINE Rx_Command   (* structured text *)
   //get input from EtherNet Adapter Module (NAP)
   
   
END_ROUTINE

ROUTINE Simulate_B_Pres0   (* structured text *)
   /*B_Pres0.CurrentValue := 3500 - CountOfTimerCompletion*60; //3440, 3380,....,0; 60/sec
   TONR(SIMULATOR);
   SIMULATOR.PRE := 1000;
   SIMULATOR.TimerEnable := 1;
   SIMULATOR.Reset := 0;
   
   if SIMULATOR.DN then
   	CTUD(CountOfTimerCompletion);
   	SIMULATOR.Reset := 1;
   end_if;
   */
END_ROUTINE

ROUTINE Update_B_Pres0   (* structured text *)
// Routine for Brakes Pressure Sensor #0
   case B_Pres0.Count of
   	0: B_Pres0.PreviousValue0 := B_Pres0.CurrentValue;
   	1: B_Pres0.PreviousValue1 := B_Pres0.CurrentValue;
   	2: B_Pres0.PreviousValue2 := B_Pres0.CurrentValue;
   	3: B_Pres0.PreviousValue3 := B_Pres0.CurrentValue;
   	4: B_Pres0.PreviousValue4 := B_Pres0.CurrentValue;
   	5: B_Pres0.PreviousValue5 := B_Pres0.CurrentValue;
   	6: B_Pres0.PreviousValue6 := B_Pres0.CurrentValue;
   	7: B_Pres0.PreviousValue7 := B_Pres0.CurrentValue;
   	8: B_Pres0.PreviousValue8 := B_Pres0.CurrentValue;
   	9: B_Pres0.PreviousValue9 := B_Pres0.CurrentValue;
   end_case;
   B_Pres0.Count := B_Pres0.Count + 1;
   if B_Pres0.Count = 10 then
   	B_Pres0.Count := 0;
   	B_Pres0.MeanStart := 1;
   end_if;
   B_Pres0.CurrentValue := Local:1:I.Ch00.Data;
   if B_Pres0.MeanStart then
   	B_Pres0.Mean10 := (B_Pres0.PreviousValue0 + B_Pres0.PreviousValue1 + B_Pres0.PreviousValue2 + B_Pres0.PreviousValue3 + B_Pres0.PreviousValue4 + B_Pres0.PreviousValue5 + B_Pres0.PreviousValue6 + B_Pres0.PreviousValue7 + B_Pres0.PreviousValue8 + B_Pres0.PreviousValue9)/10;
   	B_Pres0.StanDev := SQRT(((B_Pres0.PreviousValue0 - B_Pres0.Mean10)**2 + (B_Pres0.PreviousValue1 - B_Pres0.Mean10)**2 + (B_Pres0.PreviousValue2 - B_Pres0.Mean10)**2 + (B_Pres0.PreviousValue3 - B_Pres0.Mean10)**2 + (B_Pres0.PreviousValue4 - B_Pres0.Mean10)**2 + (B_Pres0.PreviousValue5 - B_Pres0.Mean10)**2 + (B_Pres0.PreviousValue6 - B_Pres0.Mean10)**2 + (B_Pres0.PreviousValue7 - B_Pres0.Mean10)**2 + (B_Pres0.PreviousValue8 - B_Pres0.Mean10)**2 + (B_Pres0.PreviousValue9 - B_Pres0.Mean10)**2)/10);
   end_if;
END_ROUTINE

ROUTINE Update_B_Pres1   (* structured text *)
   case B_Pres1.Count of
   	0: B_Pres1.PreviousValue0 := B_Pres1.CurrentValue;
   	1: B_Pres1.PreviousValue1 := B_Pres1.CurrentValue;
   	2: B_Pres1.PreviousValue2 := B_Pres1.CurrentValue;
   	3: B_Pres1.PreviousValue3 := B_Pres1.CurrentValue;
   	4: B_Pres1.PreviousValue4 := B_Pres1.CurrentValue;
   	5: B_Pres1.PreviousValue5 := B_Pres1.CurrentValue;
   	6: B_Pres1.PreviousValue6 := B_Pres1.CurrentValue;
   	7: B_Pres1.PreviousValue7 := B_Pres1.CurrentValue;
   	8: B_Pres1.PreviousValue8 := B_Pres1.CurrentValue;
   	9: B_Pres1.PreviousValue9 := B_Pres1.CurrentValue;
   end_case;
   B_Pres1.Count := B_Pres1.Count + 1;
   if B_Pres1.Count = 10 then
   	B_Pres1.Count := 0;
   	B_Pres1.MeanStart := 1;
   end_if;
   B_Pres1.CurrentValue := Local:1:I.Ch01.Data;
   if B_Pres1.MeanStart then
   	B_Pres1.Mean10 := (B_Pres1.PreviousValue0 + B_Pres1.PreviousValue1 + B_Pres1.PreviousValue2 + B_Pres1.PreviousValue3 + B_Pres1.PreviousValue4 + B_Pres1.PreviousValue5 + B_Pres1.PreviousValue6 + B_Pres1.PreviousValue7 + B_Pres1.PreviousValue8 + B_Pres1.PreviousValue9)/10;
   	B_Pres1.StanDev := SQRT(( (B_Pres1.PreviousValue0 - B_Pres1.Mean10)**2 + (B_Pres1.PreviousValue1 - B_Pres1.Mean10)**2 + (B_Pres1.PreviousValue2 - B_Pres1.Mean10)**2 + (B_Pres1.PreviousValue3 - B_Pres1.Mean10)**2 + (B_Pres1.PreviousValue4 - B_Pres1.Mean10)**2 + (B_Pres1.PreviousValue5 - B_Pres1.Mean10)**2 + (B_Pres1.PreviousValue6 - B_Pres1.Mean10)**2 + (B_Pres1.PreviousValue7 - B_Pres1.Mean10)**2 + (B_Pres1.PreviousValue8 - B_Pres1.Mean10)**2 + (B_Pres1.PreviousValue9 - B_Pres1.Mean10)**2)/10);
   end_if;
END_ROUTINE

ROUTINE Update_B_Pres2   (* structured text *)
   case B_Pres2.Count of
   	0: B_Pres2.PreviousValue0 := B_Pres2.CurrentValue;
   	1: B_Pres2.PreviousValue1 := B_Pres2.CurrentValue;
   	2: B_Pres2.PreviousValue2 := B_Pres2.CurrentValue;
   	3: B_Pres2.PreviousValue3 := B_Pres2.CurrentValue;
   	4: B_Pres2.PreviousValue4 := B_Pres2.CurrentValue;
   	5: B_Pres2.PreviousValue5 := B_Pres2.CurrentValue;
   	6: B_Pres2.PreviousValue6 := B_Pres2.CurrentValue;
   	7: B_Pres2.PreviousValue7 := B_Pres2.CurrentValue;
   	8: B_Pres2.PreviousValue8 := B_Pres2.CurrentValue;
   	9: B_Pres2.PreviousValue9 := B_Pres2.CurrentValue;
   end_case;
   B_Pres2.Count := B_Pres2.Count + 1;
   if B_Pres2.Count = 10 then
   	B_Pres2.Count := 0;
   	B_Pres2.MeanStart := 1;
   end_if;
   B_Pres2.CurrentValue := Local:1:I.Ch02.Data;
   if B_Pres2.MeanStart then
   	B_Pres2.Mean10 := (B_Pres2.PreviousValue0 + B_Pres2.PreviousValue1 + B_Pres2.PreviousValue2 + B_Pres2.PreviousValue3 + B_Pres2.PreviousValue4 + B_Pres2.PreviousValue5 + B_Pres2.PreviousValue6 + B_Pres2.PreviousValue7 + B_Pres2.PreviousValue8 + B_Pres2.PreviousValue9)/10;
   	B_Pres2.StanDev := SQRT(((B_Pres2.PreviousValue0 - B_Pres2.Mean10)**2 + (B_Pres2.PreviousValue1 - B_Pres2.Mean10)**2 + (B_Pres2.PreviousValue2 - B_Pres2.Mean10)**2 + (B_Pres2.PreviousValue3 - B_Pres2.Mean10)**2 + (B_Pres2.PreviousValue4 - B_Pres2.Mean10)**2 + (B_Pres2.PreviousValue5 - B_Pres2.Mean10)**2 + (B_Pres2.PreviousValue6 - B_Pres2.Mean10)**2 + (B_Pres2.PreviousValue7 - B_Pres2.Mean10)**2 + (B_Pres2.PreviousValue8 - B_Pres2.Mean10)**2 + (B_Pres2.PreviousValue9 - B_Pres2.Mean10)**2)/10);
   end_if;
END_ROUTINE

ROUTINE Update_B_Pres3   (* structured text *)
   case B_Pres3.Count of
   	0: B_Pres3.PreviousValue0 := B_Pres3.CurrentValue;
   	1: B_Pres3.PreviousValue1 := B_Pres3.CurrentValue;
   	2: B_Pres3.PreviousValue2 := B_Pres3.CurrentValue;
   	3: B_Pres3.PreviousValue3 := B_Pres3.CurrentValue;
   	4: B_Pres3.PreviousValue4 := B_Pres3.CurrentValue;
   	5: B_Pres3.PreviousValue5 := B_Pres3.CurrentValue;
   	6: B_Pres3.PreviousValue6 := B_Pres3.CurrentValue;
   	7: B_Pres3.PreviousValue7 := B_Pres3.CurrentValue;
   	8: B_Pres3.PreviousValue8 := B_Pres3.CurrentValue;
   	9: B_Pres3.PreviousValue9 := B_Pres3.CurrentValue;
   end_case;
   B_Pres3.Count := B_Pres3.Count + 1;
   if B_Pres3.Count = 10 then
   	B_Pres3.Count := 0;
   	B_Pres3.MeanStart := 1;
   end_if;
   B_Pres3.CurrentValue := Local:1:I.Ch03.Data;
   if B_Pres3.MeanStart then
   	B_Pres3.Mean10 := (B_Pres3.PreviousValue0 + B_Pres3.PreviousValue1 + B_Pres3.PreviousValue2 + B_Pres3.PreviousValue3 + B_Pres3.PreviousValue4 + B_Pres3.PreviousValue5 + B_Pres3.PreviousValue6 + B_Pres3.PreviousValue7 + B_Pres3.PreviousValue8 + B_Pres3.PreviousValue9)/10;
   	B_Pres3.StanDev := SQRT(((B_Pres3.PreviousValue0 - B_Pres3.Mean10)**2 + (B_Pres3.PreviousValue1 - B_Pres3.Mean10)**2 + (B_Pres3.PreviousValue2 - B_Pres3.Mean10)**2 + (B_Pres3.PreviousValue3 - B_Pres3.Mean10)**2 + (B_Pres3.PreviousValue4 - B_Pres3.Mean10)**2 + (B_Pres3.PreviousValue5 - B_Pres3.Mean10)**2 + (B_Pres3.PreviousValue6 - B_Pres3.Mean10)**2 + (B_Pres3.PreviousValue7 - B_Pres3.Mean10)**2 + (B_Pres3.PreviousValue8 - B_Pres3.Mean10)**2 + (B_Pres3.PreviousValue9 - B_Pres3.Mean10)**2)/10);
   end_if;
END_ROUTINE

ROUTINE Update_B_Pres4   (* structured text *)
   case B_Pres4.Count of
   	0: B_Pres4.PreviousValue0 := B_Pres4.CurrentValue;
   	1: B_Pres4.PreviousValue1 := B_Pres4.CurrentValue;
   	2: B_Pres4.PreviousValue2 := B_Pres4.CurrentValue;
   	3: B_Pres4.PreviousValue3 := B_Pres4.CurrentValue;
   	4: B_Pres4.PreviousValue4 := B_Pres4.CurrentValue;
   	5: B_Pres4.PreviousValue5 := B_Pres4.CurrentValue;
   	6: B_Pres4.PreviousValue6 := B_Pres4.CurrentValue;
   	7: B_Pres4.PreviousValue7 := B_Pres4.CurrentValue;
   	8: B_Pres4.PreviousValue8 := B_Pres4.CurrentValue;
   	9: B_Pres4.PreviousValue9 := B_Pres4.CurrentValue;
   end_case;
   B_Pres4.Count := B_Pres4.Count + 1;
   if B_Pres4.Count = 10 then
   	B_Pres4.Count := 0;
   	B_Pres4.MeanStart := 1;
   end_if;
   B_Pres4.CurrentValue := Local:1:I.Ch04.Data;
   if B_Pres4.MeanStart then
   	B_Pres4.Mean10 := (B_Pres4.PreviousValue0 + B_Pres4.PreviousValue1 + B_Pres4.PreviousValue2 + B_Pres4.PreviousValue3 + B_Pres4.PreviousValue4 + B_Pres4.PreviousValue5 + B_Pres4.PreviousValue6 + B_Pres4.PreviousValue7 + B_Pres4.PreviousValue8 + B_Pres4.PreviousValue9)/10;
   	B_Pres4.StanDev := SQRT(((B_Pres4.PreviousValue0 - B_Pres4.Mean10)**2 + (B_Pres4.PreviousValue1 - B_Pres4.Mean10)**2 + (B_Pres4.PreviousValue2 - B_Pres4.Mean10)**2 + (B_Pres4.PreviousValue3 - B_Pres4.Mean10)**2 + (B_Pres4.PreviousValue4 - B_Pres4.Mean10)**2 + (B_Pres4.PreviousValue5 - B_Pres4.Mean10)**2 + (B_Pres4.PreviousValue6 - B_Pres4.Mean10)**2 + (B_Pres4.PreviousValue7 - B_Pres4.Mean10)**2 + (B_Pres4.PreviousValue8 - B_Pres4.Mean10)**2 + (B_Pres4.PreviousValue9 - B_Pres4.Mean10)**2)/10);
   end_if;
END_ROUTINE

ROUTINE Update_B_Pres5   (* structured text *)
   case B_Pres5.Count of
   	0: B_Pres5.PreviousValue0 := B_Pres5.CurrentValue;
   	1: B_Pres5.PreviousValue1 := B_Pres5.CurrentValue;
   	2: B_Pres5.PreviousValue2 := B_Pres5.CurrentValue;
   	3: B_Pres5.PreviousValue3 := B_Pres5.CurrentValue;
   	4: B_Pres5.PreviousValue4 := B_Pres5.CurrentValue;
   	5: B_Pres5.PreviousValue5 := B_Pres5.CurrentValue;
   	6: B_Pres5.PreviousValue6 := B_Pres5.CurrentValue;
   	7: B_Pres5.PreviousValue7 := B_Pres5.CurrentValue;
   	8: B_Pres5.PreviousValue8 := B_Pres5.CurrentValue;
   	9: B_Pres5.PreviousValue9 := B_Pres5.CurrentValue;
   end_case;
   B_Pres5.Count := B_Pres5.Count + 1;
   if B_Pres5.Count = 10 then
   	B_Pres5.Count := 0;
   	B_Pres5.MeanStart := 1;
   end_if;
   B_Pres5.CurrentValue := Local:1:I.Ch05.Data;
   if B_Pres5.MeanStart then
   	B_Pres5.Mean10 := (B_Pres5.PreviousValue0 + B_Pres5.PreviousValue1 + B_Pres5.PreviousValue2 + B_Pres5.PreviousValue3 + B_Pres5.PreviousValue4 + B_Pres5.PreviousValue5 + B_Pres5.PreviousValue6 + B_Pres5.PreviousValue7 + B_Pres5.PreviousValue8 + B_Pres5.PreviousValue9)/10;
   	B_Pres5.StanDev := SQRT(((B_Pres5.PreviousValue0 - B_Pres5.Mean10)**2 + (B_Pres5.PreviousValue1 - B_Pres5.Mean10)**2 + (B_Pres5.PreviousValue2 - B_Pres5.Mean10)**2 + (B_Pres5.PreviousValue3 - B_Pres5.Mean10)**2 + (B_Pres5.PreviousValue4 - B_Pres5.Mean10)**2 + (B_Pres5.PreviousValue5 - B_Pres5.Mean10)**2 + (B_Pres5.PreviousValue6 - B_Pres5.Mean10)**2 + (B_Pres5.PreviousValue7 - B_Pres5.Mean10)**2 + (B_Pres5.PreviousValue8 - B_Pres5.Mean10)**2 + (B_Pres5.PreviousValue9 - B_Pres5.Mean10)**2)/10);
   end_if;
END_ROUTINE

ROUTINE Update_B_Pres6   (* structured text *)
   case B_Pres6.Count of
   	0: B_Pres6.PreviousValue0 := B_Pres6.CurrentValue;
   	1: B_Pres6.PreviousValue1 := B_Pres6.CurrentValue;
   	2: B_Pres6.PreviousValue2 := B_Pres6.CurrentValue;
   	3: B_Pres6.PreviousValue3 := B_Pres6.CurrentValue;
   	4: B_Pres6.PreviousValue4 := B_Pres6.CurrentValue;
   	5: B_Pres6.PreviousValue5 := B_Pres6.CurrentValue;
   	6: B_Pres6.PreviousValue6 := B_Pres6.CurrentValue;
   	7: B_Pres6.PreviousValue7 := B_Pres6.CurrentValue;
   	8: B_Pres6.PreviousValue8 := B_Pres6.CurrentValue;
   	9: B_Pres6.PreviousValue9 := B_Pres6.CurrentValue;
   end_case;
   B_Pres6.Count := B_Pres6.Count + 1;
   if B_Pres6.Count = 10 then
   	B_Pres6.Count := 0;
   	B_Pres6.MeanStart := 1;
   end_if;
   B_Pres6.CurrentValue := Local:1:I.Ch06.Data;
   if B_Pres6.MeanStart then
   	B_Pres6.Mean10 := (B_Pres6.PreviousValue0 + B_Pres6.PreviousValue1 + B_Pres6.PreviousValue2 + B_Pres6.PreviousValue3 + B_Pres6.PreviousValue4 + B_Pres6.PreviousValue5 + B_Pres6.PreviousValue6 + B_Pres6.PreviousValue7 + B_Pres6.PreviousValue8 + B_Pres6.PreviousValue9)/10;
   	B_Pres6.StanDev := SQRT(((B_Pres6.PreviousValue0 - B_Pres6.Mean10)**2 + (B_Pres6.PreviousValue1 - B_Pres6.Mean10)**2 + (B_Pres6.PreviousValue2 - B_Pres6.Mean10)**2 + (B_Pres6.PreviousValue3 - B_Pres6.Mean10)**2 + (B_Pres6.PreviousValue4 - B_Pres6.Mean10)**2 + (B_Pres6.PreviousValue5 - B_Pres6.Mean10)**2 + (B_Pres6.PreviousValue6 - B_Pres6.Mean10)**2 + (B_Pres6.PreviousValue7 - B_Pres6.Mean10)**2 + (B_Pres6.PreviousValue8 - B_Pres6.Mean10)**2 + (B_Pres6.PreviousValue9 - B_Pres6.Mean10)**2)/10);
   end_if;
END_ROUTINE

ROUTINE Update_B_Pres7   (* structured text *)
   case B_Pres7.Count of
   	0: B_Pres7.PreviousValue0 := B_Pres7.CurrentValue;
   	1: B_Pres7.PreviousValue1 := B_Pres7.CurrentValue;
   	2: B_Pres7.PreviousValue2 := B_Pres7.CurrentValue;
   	3: B_Pres7.PreviousValue3 := B_Pres7.CurrentValue;
   	4: B_Pres7.PreviousValue4 := B_Pres7.CurrentValue;
   	5: B_Pres7.PreviousValue5 := B_Pres7.CurrentValue;
   	6: B_Pres7.PreviousValue6 := B_Pres7.CurrentValue;
   	7: B_Pres7.PreviousValue7 := B_Pres7.CurrentValue;
   	8: B_Pres7.PreviousValue8 := B_Pres7.CurrentValue;
   	9: B_Pres7.PreviousValue9 := B_Pres7.CurrentValue;
   end_case;
   B_Pres7.Count := B_Pres7.Count + 1;
   if B_Pres7.Count = 10 then
   	B_Pres7.Count := 0;
   	B_Pres7.MeanStart := 1;
   end_if;
   B_Pres7.CurrentValue := Local:1:I.Ch07.Data;
   if B_Pres7.MeanStart then
   	B_Pres7.Mean10 := (B_Pres7.PreviousValue0 + B_Pres7.PreviousValue1 + B_Pres7.PreviousValue2 + B_Pres7.PreviousValue3 + B_Pres7.PreviousValue4 + B_Pres7.PreviousValue5 + B_Pres7.PreviousValue6 + B_Pres7.PreviousValue7 + B_Pres7.PreviousValue8 + B_Pres7.PreviousValue9)/10;
   	B_Pres7.StanDev := SQRT(((B_Pres7.PreviousValue0 - B_Pres7.Mean10)**2 + (B_Pres7.PreviousValue1 - B_Pres7.Mean10)**2 + (B_Pres7.PreviousValue2 - B_Pres7.Mean10)**2 + (B_Pres7.PreviousValue3 - B_Pres7.Mean10)**2 + (B_Pres7.PreviousValue4 - B_Pres7.Mean10)**2 + (B_Pres7.PreviousValue5 - B_Pres7.Mean10)**2 + (B_Pres7.PreviousValue6 - B_Pres7.Mean10)**2 + (B_Pres7.PreviousValue7 - B_Pres7.Mean10)**2 + (B_Pres7.PreviousValue8 - B_Pres7.Mean10)**2 + (B_Pres7.PreviousValue9 - B_Pres7.Mean10)**2)/10);
   end_if;
END_ROUTINE

ROUTINE Update_B_Pres8   (* structured text *)
   case B_Pres8.Count of
   	0: B_Pres8.PreviousValue0 := B_Pres8.CurrentValue;
   	1: B_Pres8.PreviousValue1 := B_Pres8.CurrentValue;
   	2: B_Pres8.PreviousValue2 := B_Pres8.CurrentValue;
   	3: B_Pres8.PreviousValue3 := B_Pres8.CurrentValue;
   	4: B_Pres8.PreviousValue4 := B_Pres8.CurrentValue;
   	5: B_Pres8.PreviousValue5 := B_Pres8.CurrentValue;
   	6: B_Pres8.PreviousValue6 := B_Pres8.CurrentValue;
   	7: B_Pres8.PreviousValue7 := B_Pres8.CurrentValue;
   	8: B_Pres8.PreviousValue8 := B_Pres8.CurrentValue;
   	9: B_Pres8.PreviousValue9 := B_Pres8.CurrentValue;
   end_case;
   B_Pres8.Count := B_Pres8.Count + 1;
   if B_Pres8.Count = 10 then
   	B_Pres8.Count := 0;
   	B_Pres8.MeanStart := 1;
   end_if;
   B_Pres8.CurrentValue := Local:2:I.Ch00.Data;
   if B_Pres8.MeanStart then
   	B_Pres8.Mean10 := (B_Pres8.PreviousValue0 + B_Pres8.PreviousValue1 + B_Pres8.PreviousValue2 + B_Pres8.PreviousValue3 + B_Pres8.PreviousValue4 + B_Pres8.PreviousValue5 + B_Pres8.PreviousValue6 + B_Pres8.PreviousValue7 + B_Pres8.PreviousValue8 + B_Pres8.PreviousValue9)/10;
   	B_Pres8.StanDev := SQRT(((B_Pres8.PreviousValue0 - B_Pres8.Mean10)**2 + (B_Pres8.PreviousValue1 - B_Pres8.Mean10)**2 + (B_Pres8.PreviousValue2 - B_Pres8.Mean10)**2 + (B_Pres8.PreviousValue3 - B_Pres8.Mean10)**2 + (B_Pres8.PreviousValue4 - B_Pres8.Mean10)**2 + (B_Pres8.PreviousValue5 - B_Pres8.Mean10)**2 + (B_Pres8.PreviousValue6 - B_Pres8.Mean10)**2 + (B_Pres8.PreviousValue7 - B_Pres8.Mean10)**2 + (B_Pres8.PreviousValue8 - B_Pres8.Mean10)**2 + (B_Pres8.PreviousValue9 - B_Pres8.Mean10)**2)/10);
   end_if;
END_ROUTINE

ROUTINE Update_B_Pres9   (* structured text *)
   case B_Pres9.Count of
   	0: B_Pres9.PreviousValue0 := B_Pres9.CurrentValue;
   	1: B_Pres9.PreviousValue1 := B_Pres9.CurrentValue;
   	2: B_Pres9.PreviousValue2 := B_Pres9.CurrentValue;
   	3: B_Pres9.PreviousValue3 := B_Pres9.CurrentValue;
   	4: B_Pres9.PreviousValue4 := B_Pres9.CurrentValue;
   	5: B_Pres9.PreviousValue5 := B_Pres9.CurrentValue;
   	6: B_Pres9.PreviousValue6 := B_Pres9.CurrentValue;
   	7: B_Pres9.PreviousValue7 := B_Pres9.CurrentValue;
   	8: B_Pres9.PreviousValue8 := B_Pres9.CurrentValue;
   	9: B_Pres9.PreviousValue9 := B_Pres9.CurrentValue;
   end_case;
   B_Pres9.Count := B_Pres9.Count + 1;
   if B_Pres9.Count = 10 then
   	B_Pres9.Count := 0;
   	B_Pres9.MeanStart := 1;
   end_if;
   B_Pres9.CurrentValue := Local:2:I.Ch01.Data;
   if B_Pres9.MeanStart then
   	B_Pres9.Mean10 := (B_Pres9.PreviousValue0 + B_Pres9.PreviousValue1 + B_Pres9.PreviousValue2 + B_Pres9.PreviousValue3 + B_Pres9.PreviousValue4 + B_Pres9.PreviousValue5 + B_Pres9.PreviousValue6 + B_Pres9.PreviousValue7 + B_Pres9.PreviousValue8 + B_Pres9.PreviousValue9)/10;
   	B_Pres9.StanDev := SQRT(((B_Pres9.PreviousValue0 - B_Pres9.Mean10)**2 + (B_Pres9.PreviousValue1 - B_Pres9.Mean10)**2 + (B_Pres9.PreviousValue2 - B_Pres9.Mean10)**2 + (B_Pres9.PreviousValue3 - B_Pres9.Mean10)**2 + (B_Pres9.PreviousValue4 - B_Pres9.Mean10)**2 + (B_Pres9.PreviousValue5 - B_Pres9.Mean10)**2 + (B_Pres9.PreviousValue6 - B_Pres9.Mean10)**2 + (B_Pres9.PreviousValue7 - B_Pres9.Mean10)**2 + (B_Pres9.PreviousValue8 - B_Pres9.Mean10)**2 + (B_Pres9.PreviousValue9 - B_Pres9.Mean10)**2)/10);
   end_if;
END_ROUTINE

ROUTINE Update_B_Tem0   (* structured text *)
   case B_Tem0.Count of
   	0: B_Tem0.PreviousValue0 := B_Tem0.CurrentValue;
   	1: B_Tem0.PreviousValue1 := B_Tem0.CurrentValue;
   	2: B_Tem0.PreviousValue2 := B_Tem0.CurrentValue;
   	3: B_Tem0.PreviousValue3 := B_Tem0.CurrentValue;
   	4: B_Tem0.PreviousValue4 := B_Tem0.CurrentValue;
   	5: B_Tem0.PreviousValue5 := B_Tem0.CurrentValue;
   	6: B_Tem0.PreviousValue6 := B_Tem0.CurrentValue;
   	7: B_Tem0.PreviousValue7 := B_Tem0.CurrentValue;
   	8: B_Tem0.PreviousValue8 := B_Tem0.CurrentValue;
   	9: B_Tem0.PreviousValue9 := B_Tem0.CurrentValue;
   end_case;
   B_Tem0.Count := B_Tem0.Count + 1;
   if B_Tem0.Count = 10 then
   	B_Tem0.Count := 0;
   	B_Tem0.MeanStart := 1;
   end_if;
   B_Tem0.CurrentValue := Local:2:I.Ch02.Data;
   if B_Tem0.MeanStart then
   	B_Tem0.Mean10 := (B_Tem0.PreviousValue0 + B_Tem0.PreviousValue1 + B_Tem0.PreviousValue2 + B_Tem0.PreviousValue3 + B_Tem0.PreviousValue4 + B_Tem0.PreviousValue5 + B_Tem0.PreviousValue6 + B_Tem0.PreviousValue7 + B_Tem0.PreviousValue8 + B_Tem0.PreviousValue9)/10;
   	B_Tem0.StanDev := SQRT(((B_Tem0.PreviousValue0 - B_Tem0.Mean10)**2 + (B_Tem0.PreviousValue1 - B_Tem0.Mean10)**2 + (B_Tem0.PreviousValue2 - B_Tem0.Mean10)**2 + (B_Tem0.PreviousValue3 - B_Tem0.Mean10)**2 + (B_Tem0.PreviousValue4 - B_Tem0.Mean10)**2 + (B_Tem0.PreviousValue5 - B_Tem0.Mean10)**2 + (B_Tem0.PreviousValue6 - B_Tem0.Mean10)**2 + (B_Tem0.PreviousValue7 - B_Tem0.Mean10)**2 + (B_Tem0.PreviousValue8 - B_Tem0.Mean10)**2 + (B_Tem0.PreviousValue9 - B_Tem0.Mean10)**2)/10);
   end_if;
END_ROUTINE

ROUTINE Update_B_Tem1   (* structured text *)
   case B_Tem1.Count of
   	0: B_Tem1.PreviousValue0 := B_Tem1.CurrentValue;
   	1: B_Tem1.PreviousValue1 := B_Tem1.CurrentValue;
   	2: B_Tem1.PreviousValue2 := B_Tem1.CurrentValue;
   	3: B_Tem1.PreviousValue3 := B_Tem1.CurrentValue;
   	4: B_Tem1.PreviousValue4 := B_Tem1.CurrentValue;
   	5: B_Tem1.PreviousValue5 := B_Tem1.CurrentValue;
   	6: B_Tem1.PreviousValue6 := B_Tem1.CurrentValue;
   	7: B_Tem1.PreviousValue7 := B_Tem1.CurrentValue;
   	8: B_Tem1.PreviousValue8 := B_Tem1.CurrentValue;
   	9: B_Tem1.PreviousValue9 := B_Tem1.CurrentValue;
   end_case;
   B_Tem1.Count := B_Tem1.Count + 1;
   if B_Tem1.Count = 10 then
   	B_Tem1.Count := 0;
   	B_Tem1.MeanStart := 1;
   end_if;
   B_Tem1.CurrentValue := Local:2:I.Ch03.Data;
   if B_Tem1.MeanStart then
   	B_Tem1.Mean10 := (B_Tem1.PreviousValue0 + B_Tem1.PreviousValue1 + B_Tem1.PreviousValue2 + B_Tem1.PreviousValue3 + B_Tem1.PreviousValue4 + B_Tem1.PreviousValue5 + B_Tem1.PreviousValue6 + B_Tem1.PreviousValue7 + B_Tem1.PreviousValue8 + B_Tem1.PreviousValue9)/10;
   	B_Tem1.StanDev := SQRT(((B_Tem1.PreviousValue0 - B_Tem1.Mean10)**2 + (B_Tem1.PreviousValue1 - B_Tem1.Mean10)**2 + (B_Tem1.PreviousValue2 - B_Tem1.Mean10)**2 + (B_Tem1.PreviousValue3 - B_Tem1.Mean10)**2 + (B_Tem1.PreviousValue4 - B_Tem1.Mean10)**2 + (B_Tem1.PreviousValue5 - B_Tem1.Mean10)**2 + (B_Tem1.PreviousValue6 - B_Tem1.Mean10)**2 + (B_Tem1.PreviousValue7 - B_Tem1.Mean10)**2 + (B_Tem1.PreviousValue8 - B_Tem1.Mean10)**2 + (B_Tem1.PreviousValue9 - B_Tem1.Mean10)**2)/10);
   end_if;
END_ROUTINE

ROUTINE Update_Bat_Current   (* structured text *)
   //BMS to PLC, RS485 communication
END_ROUTINE

ROUTINE Update_Bat_Temp   (* structured text *)
   //BMS to PLC, RS485 communication
END_ROUTINE

ROUTINE Update_Bat_Voltage   (* structured text *)
   //BMS to PLC, RS485 communication
END_ROUTINE

ROUTINE Update_C_Las0   (* structured text *)
   case C_Las0.Count of
   	0: C_Las0.PreviousValue0 := C_Las0.CurrentValue;
   	1: C_Las0.PreviousValue1 := C_Las0.CurrentValue;
   	2: C_Las0.PreviousValue2 := C_Las0.CurrentValue;
   	3: C_Las0.PreviousValue3 := C_Las0.CurrentValue;
   	4: C_Las0.PreviousValue4 := C_Las0.CurrentValue;
   	5: C_Las0.PreviousValue5 := C_Las0.CurrentValue;
   	6: C_Las0.PreviousValue6 := C_Las0.CurrentValue;
   	7: C_Las0.PreviousValue7 := C_Las0.CurrentValue;
   	8: C_Las0.PreviousValue8 := C_Las0.CurrentValue;
   	9: C_Las0.PreviousValue9 := C_Las0.CurrentValue;
   end_case;
   C_Las0.Count := C_Las0.Count + 1;
   if C_Las0.Count = 10 then
   	C_Las0.Count := 0;
   	C_Las0.MeanStart := 1;
   end_if;
   C_Las0.CurrentValue := Local:7:I.Counter00.Count;
   if C_Las0.MeanStart then
   	C_Las0.Mean10 := (C_Las0.PreviousValue0 + C_Las0.PreviousValue1 + C_Las0.PreviousValue2 + C_Las0.PreviousValue3 + C_Las0.PreviousValue4 + C_Las0.PreviousValue5 + C_Las0.PreviousValue6 + C_Las0.PreviousValue7 + C_Las0.PreviousValue8 + C_Las0.PreviousValue9)/10;
   	C_Las0.StanDev := SQRT(((C_Las0.PreviousValue0 - C_Las0.Mean10)**2 + (C_Las0.PreviousValue1 - C_Las0.Mean10)**2 + (C_Las0.PreviousValue2 - C_Las0.Mean10)**2 + (C_Las0.PreviousValue3 - C_Las0.Mean10)**2 + (C_Las0.PreviousValue4 - C_Las0.Mean10)**2 + (C_Las0.PreviousValue5 - C_Las0.Mean10)**2 + (C_Las0.PreviousValue6 - C_Las0.Mean10)**2 + (C_Las0.PreviousValue7 - C_Las0.Mean10)**2 + (C_Las0.PreviousValue8 - C_Las0.Mean10)**2 + (C_Las0.PreviousValue9 - C_Las0.Mean10)**2)/10);
   end_if;
END_ROUTINE

ROUTINE Update_C_Las1   (* structured text *)
   case C_Las1.Count of
   	0: C_Las1.PreviousValue0 := C_Las1.CurrentValue;
   	1: C_Las1.PreviousValue1 := C_Las1.CurrentValue;
   	2: C_Las1.PreviousValue2 := C_Las1.CurrentValue;
   	3: C_Las1.PreviousValue3 := C_Las1.CurrentValue;
   	4: C_Las1.PreviousValue4 := C_Las1.CurrentValue;
   	5: C_Las1.PreviousValue5 := C_Las1.CurrentValue;
   	6: C_Las1.PreviousValue6 := C_Las1.CurrentValue;
   	7: C_Las1.PreviousValue7 := C_Las1.CurrentValue;
   	8: C_Las1.PreviousValue8 := C_Las1.CurrentValue;
   	9: C_Las1.PreviousValue9 := C_Las1.CurrentValue;
   end_case;
   C_Las1.Count := C_Las1.Count + 1;
   if C_Las1.Count = 10 then
   	C_Las1.Count := 0;
   	C_Las1.MeanStart := 1;
   end_if;
   C_Las1.CurrentValue := Local:7:I.Counter01.Count;
   if C_Las1.MeanStart then
   	C_Las1.Mean10 := (C_Las1.PreviousValue0 + C_Las1.PreviousValue1 + C_Las1.PreviousValue2 + C_Las1.PreviousValue3 + C_Las1.PreviousValue4 + C_Las1.PreviousValue5 + C_Las1.PreviousValue6 + C_Las1.PreviousValue7 + C_Las1.PreviousValue8 + C_Las1.PreviousValue9)/10;
   	C_Las1.StanDev := SQRT(((C_Las1.PreviousValue0 - C_Las1.Mean10)**2 + (C_Las1.PreviousValue1 - C_Las1.Mean10)**2 + (C_Las1.PreviousValue2 - C_Las1.Mean10)**2 + (C_Las1.PreviousValue3 - C_Las1.Mean10)**2 + (C_Las1.PreviousValue4 - C_Las1.Mean10)**2 + (C_Las1.PreviousValue5 - C_Las1.Mean10)**2 + (C_Las1.PreviousValue6 - C_Las1.Mean10)**2 + (C_Las1.PreviousValue7 - C_Las1.Mean10)**2 + (C_Las1.PreviousValue8 - C_Las1.Mean10)**2 + (C_Las1.PreviousValue9 - C_Las1.Mean10)**2)/10);
   end_if;
END_ROUTINE

ROUTINE Update_P_Pres0   (* structured text *)
   case P_Pres0.Count of
   	0: P_Pres0.PreviousValue0 := P_Pres0.CurrentValue;
   	1: P_Pres0.PreviousValue1 := P_Pres0.CurrentValue;
   	2: P_Pres0.PreviousValue2 := P_Pres0.CurrentValue;
   	3: P_Pres0.PreviousValue3 := P_Pres0.CurrentValue;
   	4: P_Pres0.PreviousValue4 := P_Pres0.CurrentValue;
   	5: P_Pres0.PreviousValue5 := P_Pres0.CurrentValue;
   	6: P_Pres0.PreviousValue6 := P_Pres0.CurrentValue;
   	7: P_Pres0.PreviousValue7 := P_Pres0.CurrentValue;
   	8: P_Pres0.PreviousValue8 := P_Pres0.CurrentValue;
   	9: P_Pres0.PreviousValue9 := P_Pres0.CurrentValue;
   end_case;
   P_Pres0.Count := P_Pres0.Count + 1;
   if P_Pres0.Count = 10 then
   	P_Pres0.Count := 0;
   	P_Pres0.MeanStart := 1;
   end_if;
   P_Pres0.CurrentValue := Local:3:I.Ch00.Data;
   if P_Pres0.MeanStart then
   	P_Pres0.Mean10 := (P_Pres0.PreviousValue0 + P_Pres0.PreviousValue1 + P_Pres0.PreviousValue2 + P_Pres0.PreviousValue3 + P_Pres0.PreviousValue4 + P_Pres0.PreviousValue5 + P_Pres0.PreviousValue6 + P_Pres0.PreviousValue7 + P_Pres0.PreviousValue8 + P_Pres0.PreviousValue9)/10;
   	P_Pres0.StanDev := SQRT(((P_Pres0.PreviousValue0 - P_Pres0.Mean10)**2 + (P_Pres0.PreviousValue1 - P_Pres0.Mean10)**2 + (P_Pres0.PreviousValue2 - P_Pres0.Mean10)**2 + (P_Pres0.PreviousValue3 - P_Pres0.Mean10)**2 + (P_Pres0.PreviousValue4 - P_Pres0.Mean10)**2 + (P_Pres0.PreviousValue5 - P_Pres0.Mean10)**2 + (P_Pres0.PreviousValue6 - P_Pres0.Mean10)**2 + (P_Pres0.PreviousValue7 - P_Pres0.Mean10)**2 + (P_Pres0.PreviousValue8 - P_Pres0.Mean10)**2 + (P_Pres0.PreviousValue9 - P_Pres0.Mean10)**2)/10);
   end_if;
END_ROUTINE

ROUTINE Update_P_Pres1   (* structured text *)
   case P_Pres1.Count of
   	0: P_Pres1.PreviousValue0 := P_Pres1.CurrentValue;
   	1: P_Pres1.PreviousValue1 := P_Pres1.CurrentValue;
   	2: P_Pres1.PreviousValue2 := P_Pres1.CurrentValue;
   	3: P_Pres1.PreviousValue3 := P_Pres1.CurrentValue;
   	4: P_Pres1.PreviousValue4 := P_Pres1.CurrentValue;
   	5: P_Pres1.PreviousValue5 := P_Pres1.CurrentValue;
   	6: P_Pres1.PreviousValue6 := P_Pres1.CurrentValue;
   	7: P_Pres1.PreviousValue7 := P_Pres1.CurrentValue;
   	8: P_Pres1.PreviousValue8 := P_Pres1.CurrentValue;
   	9: P_Pres1.PreviousValue9 := P_Pres1.CurrentValue;
   end_case;
   P_Pres1.Count := P_Pres1.Count + 1;
   if P_Pres1.Count = 10 then
   	P_Pres1.Count := 0;
   	P_Pres0.MeanStart := 1;
   end_if;
   P_Pres1.CurrentValue := Local:3:I.Ch01.Data;
   if P_Pres1.MeanStart then
   	P_Pres1.Mean10 := (P_Pres1.PreviousValue0 + P_Pres1.PreviousValue1 + P_Pres1.PreviousValue2 + P_Pres1.PreviousValue3 + P_Pres1.PreviousValue4 + P_Pres1.PreviousValue5 + P_Pres1.PreviousValue6 + P_Pres1.PreviousValue7 + P_Pres1.PreviousValue8 + P_Pres1.PreviousValue9)/10;
   	P_Pres1.StanDev := SQRT(((P_Pres1.PreviousValue0 - P_Pres1.Mean10)**2 + (P_Pres1.PreviousValue1 - P_Pres1.Mean10)**2 + (P_Pres1.PreviousValue2 - P_Pres1.Mean10)**2 + (P_Pres1.PreviousValue3 - P_Pres1.Mean10)**2 + (P_Pres1.PreviousValue4 - P_Pres1.Mean10)**2 + (P_Pres1.PreviousValue5 - P_Pres1.Mean10)**2 + (P_Pres1.PreviousValue6 - P_Pres1.Mean10)**2 + (P_Pres1.PreviousValue7 - P_Pres1.Mean10)**2 + (P_Pres1.PreviousValue8 - P_Pres1.Mean10)**2 + (P_Pres1.PreviousValue9 - P_Pres1.Mean10)**2)/10);
   end_if;
END_ROUTINE

ROUTINE Update_P_Pres2   (* structured text *)
   case P_Pres2.Count of
   	0: P_Pres2.PreviousValue0 := P_Pres2.CurrentValue;
   	1: P_Pres2.PreviousValue1 := P_Pres2.CurrentValue;
   	2: P_Pres2.PreviousValue2 := P_Pres2.CurrentValue;
   	3: P_Pres2.PreviousValue3 := P_Pres2.CurrentValue;
   	4: P_Pres2.PreviousValue4 := P_Pres2.CurrentValue;
   	5: P_Pres2.PreviousValue5 := P_Pres2.CurrentValue;
   	6: P_Pres2.PreviousValue6 := P_Pres2.CurrentValue;
   	7: P_Pres2.PreviousValue7 := P_Pres2.CurrentValue;
   	8: P_Pres2.PreviousValue8 := P_Pres2.CurrentValue;
   	9: P_Pres2.PreviousValue9 := P_Pres2.CurrentValue;
   end_case;
   P_Pres2.Count := P_Pres2.Count + 1;
   if P_Pres2.Count = 10 then
   	P_Pres2.Count := 0;
   	P_Pres2.MeanStart := 1;
   end_if;
   P_Pres2.CurrentValue := Local:3:I.Ch02.Data;
   if P_Pres2.MeanStart then
   	P_Pres2.Mean10 := (P_Pres2.PreviousValue0 + P_Pres2.PreviousValue1 + P_Pres2.PreviousValue2 + P_Pres2.PreviousValue3 + P_Pres2.PreviousValue4 + P_Pres2.PreviousValue5 + P_Pres2.PreviousValue6 + P_Pres2.PreviousValue7 + P_Pres2.PreviousValue8 + P_Pres2.PreviousValue9)/10;
   	P_Pres2.StanDev := SQRT(((P_Pres2.PreviousValue0 - P_Pres2.Mean10)**2 + (P_Pres2.PreviousValue1 - P_Pres2.Mean10)**2 + (P_Pres2.PreviousValue2 - P_Pres2.Mean10)**2 + (P_Pres2.PreviousValue3 - P_Pres2.Mean10)**2 + (P_Pres2.PreviousValue4 - P_Pres2.Mean10)**2 + (P_Pres2.PreviousValue5 - P_Pres2.Mean10)**2 + (P_Pres2.PreviousValue6 - P_Pres2.Mean10)**2 + (P_Pres2.PreviousValue7 - P_Pres2.Mean10)**2 + (P_Pres2.PreviousValue8 - P_Pres2.Mean10)**2 + (P_Pres2.PreviousValue9 - P_Pres2.Mean10)**2)/10);
   end_if;
END_ROUTINE

ROUTINE Update_P_Pres3   (* structured text *)
   case P_Pres3.Count of
   	0: P_Pres3.PreviousValue0 := P_Pres3.CurrentValue;
   	1: P_Pres3.PreviousValue1 := P_Pres3.CurrentValue;
   	2: P_Pres3.PreviousValue2 := P_Pres3.CurrentValue;
   	3: P_Pres3.PreviousValue3 := P_Pres3.CurrentValue;
   	4: P_Pres3.PreviousValue4 := P_Pres3.CurrentValue;
   	5: P_Pres3.PreviousValue5 := P_Pres3.CurrentValue;
   	6: P_Pres3.PreviousValue6 := P_Pres3.CurrentValue;
   	7: P_Pres3.PreviousValue7 := P_Pres3.CurrentValue;
   	8: P_Pres3.PreviousValue8 := P_Pres3.CurrentValue;
   	9: P_Pres3.PreviousValue9 := P_Pres3.CurrentValue;
   end_case;
   P_Pres3.Count := P_Pres3.Count + 1;
   if P_Pres3.Count = 10 then
   	P_Pres3.Count := 0;
   	P_Pres3.MeanStart := 1;
   end_if;
   P_Pres3.CurrentValue := Local:3:I.Ch03.Data;
   if P_Pres3.MeanStart then
   	P_Pres3.Mean10 := (P_Pres3.PreviousValue0 + P_Pres3.PreviousValue1 + P_Pres3.PreviousValue2 + P_Pres3.PreviousValue3 + P_Pres3.PreviousValue4 + P_Pres3.PreviousValue5 + P_Pres3.PreviousValue6 + P_Pres3.PreviousValue7 + P_Pres3.PreviousValue8 + P_Pres3.PreviousValue9)/10;
   	P_Pres3.StanDev := SQRT(((P_Pres3.PreviousValue0 - P_Pres3.Mean10)**2 + (P_Pres3.PreviousValue1 - P_Pres3.Mean10)**2 + (P_Pres3.PreviousValue2 - P_Pres3.Mean10)**2 + (P_Pres3.PreviousValue3 - P_Pres3.Mean10)**2 + (P_Pres3.PreviousValue4 - P_Pres3.Mean10)**2 + (P_Pres3.PreviousValue5 - P_Pres3.Mean10)**2 + (P_Pres3.PreviousValue6 - P_Pres3.Mean10)**2 + (P_Pres3.PreviousValue7 - P_Pres3.Mean10)**2 + (P_Pres3.PreviousValue8 - P_Pres3.Mean10)**2 + (P_Pres3.PreviousValue9 - P_Pres3.Mean10)**2)/10);
   end_if;
END_ROUTINE

ROUTINE Update_P_Pres4   (* structured text *)
   case P_Pres4.Count of
   	0: P_Pres4.PreviousValue0 := P_Pres4.CurrentValue;
   	1: P_Pres4.PreviousValue1 := P_Pres4.CurrentValue;
   	2: P_Pres4.PreviousValue2 := P_Pres4.CurrentValue;
   	3: P_Pres4.PreviousValue3 := P_Pres4.CurrentValue;
   	4: P_Pres4.PreviousValue4 := P_Pres4.CurrentValue;
   	5: P_Pres4.PreviousValue5 := P_Pres4.CurrentValue;
   	6: P_Pres4.PreviousValue6 := P_Pres4.CurrentValue;
   	7: P_Pres4.PreviousValue7 := P_Pres4.CurrentValue;
   	8: P_Pres4.PreviousValue8 := P_Pres4.CurrentValue;
   	9: P_Pres4.PreviousValue9 := P_Pres4.CurrentValue;
   end_case;
   P_Pres4.Count := P_Pres4.Count + 1;
   if P_Pres4.Count = 10 then
   	P_Pres4.Count := 0;
   	P_Pres4.MeanStart := 1;
   end_if;
   P_Pres4.CurrentValue := Local:3:I.Ch04.Data;
   if P_Pres4.MeanStart then
   	P_Pres4.Mean10 := (P_Pres4.PreviousValue0 + P_Pres4.PreviousValue1 + P_Pres4.PreviousValue2 + P_Pres4.PreviousValue3 + P_Pres4.PreviousValue4 + P_Pres4.PreviousValue5 + P_Pres4.PreviousValue6 + P_Pres4.PreviousValue7 + P_Pres4.PreviousValue8 + P_Pres4.PreviousValue9)/10;
   	P_Pres4.StanDev := SQRT(((P_Pres4.PreviousValue0 - P_Pres4.Mean10)**2 + (P_Pres4.PreviousValue1 - P_Pres4.Mean10)**2 + (P_Pres4.PreviousValue2 - P_Pres4.Mean10)**2 + (P_Pres4.PreviousValue3 - P_Pres4.Mean10)**2 + (P_Pres4.PreviousValue4 - P_Pres4.Mean10)**2 + (P_Pres4.PreviousValue5 - P_Pres4.Mean10)**2 + (P_Pres4.PreviousValue6 - P_Pres4.Mean10)**2 + (P_Pres4.PreviousValue7 - P_Pres4.Mean10)**2 + (P_Pres4.PreviousValue8 - P_Pres4.Mean10)**2 + (P_Pres4.PreviousValue9 - P_Pres4.Mean10)**2)/10);
   end_if;
END_ROUTINE

ROUTINE Update_P_Tem0   (* structured text *)
   case P_Tem0.Count of
   	0: P_Tem0.PreviousValue0 := P_Tem0.CurrentValue;
   	1: P_Tem0.PreviousValue1 := P_Tem0.CurrentValue;
   	2: P_Tem0.PreviousValue2 := P_Tem0.CurrentValue;
   	3: P_Tem0.PreviousValue3 := P_Tem0.CurrentValue;
   	4: P_Tem0.PreviousValue4 := P_Tem0.CurrentValue;
   	5: P_Tem0.PreviousValue5 := P_Tem0.CurrentValue;
   	6: P_Tem0.PreviousValue6 := P_Tem0.CurrentValue;
   	7: P_Tem0.PreviousValue7 := P_Tem0.CurrentValue;
   	8: P_Tem0.PreviousValue8 := P_Tem0.CurrentValue;
   	9: P_Tem0.PreviousValue9 := P_Tem0.CurrentValue;
   end_case;
   P_Tem0.Count := P_Tem0.Count + 1;
   if P_Tem0.Count = 10 then
   	P_Tem0.Count := 0;
   	P_Tem0.MeanStart := 1;
   end_if;
   P_Tem0.CurrentValue := Local:3:I.Ch05.Data;
   if P_Tem0.MeanStart then
   	P_Tem0.Mean10 := (P_Tem0.PreviousValue0 + P_Tem0.PreviousValue1 + P_Tem0.PreviousValue2 + P_Tem0.PreviousValue3 + P_Tem0.PreviousValue4 + P_Tem0.PreviousValue5 + P_Tem0.PreviousValue6 + P_Tem0.PreviousValue7 + P_Tem0.PreviousValue8 + P_Tem0.PreviousValue9)/10;
   	P_Tem0.StanDev := SQRT(((P_Tem0.PreviousValue0 - P_Tem0.Mean10)**2 + (P_Tem0.PreviousValue1 - P_Tem0.Mean10)**2 + (P_Tem0.PreviousValue2 - P_Tem0.Mean10)**2 + (P_Tem0.PreviousValue3 - P_Tem0.Mean10)**2 + (P_Tem0.PreviousValue4 - P_Tem0.Mean10)**2 + (P_Tem0.PreviousValue5 - P_Tem0.Mean10)**2 + (P_Tem0.PreviousValue6 - P_Tem0.Mean10)**2 + (P_Tem0.PreviousValue7 - P_Tem0.Mean10)**2 + (P_Tem0.PreviousValue8 - P_Tem0.Mean10)**2 + (P_Tem0.PreviousValue9 - P_Tem0.Mean10)**2)/10);
   end_if;
END_ROUTINE

ROUTINE Update_P_Tem1   (* structured text *)
   case P_Tem1.Count of
   	0: P_Tem1.PreviousValue0 := P_Tem1.CurrentValue;
   	1: P_Tem1.PreviousValue1 := P_Tem1.CurrentValue;
   	2: P_Tem1.PreviousValue2 := P_Tem1.CurrentValue;
   	3: P_Tem1.PreviousValue3 := P_Tem1.CurrentValue;
   	4: P_Tem1.PreviousValue4 := P_Tem1.CurrentValue;
   	5: P_Tem1.PreviousValue5 := P_Tem1.CurrentValue;
   	6: P_Tem1.PreviousValue6 := P_Tem1.CurrentValue;
   	7: P_Tem1.PreviousValue7 := P_Tem1.CurrentValue;
   	8: P_Tem1.PreviousValue8 := P_Tem1.CurrentValue;
   	9: P_Tem1.PreviousValue9 := P_Tem1.CurrentValue;
   end_case;
   P_Tem1.Count := P_Tem1.Count + 1;
   if P_Tem1.Count = 10 then
   	P_Tem1.Count := 0;
   	P_Tem1.MeanStart := 1;
   end_if;
   P_Tem1.CurrentValue := Local:3:I.Ch06.Data;
   if P_Tem1.MeanStart then
   	P_Tem1.Mean10 := (P_Tem1.PreviousValue0 + P_Tem1.PreviousValue1 + P_Tem1.PreviousValue2 + P_Tem1.PreviousValue3 + P_Tem1.PreviousValue4 + P_Tem1.PreviousValue5 + P_Tem1.PreviousValue6 + P_Tem1.PreviousValue7 + P_Tem1.PreviousValue8 + P_Tem1.PreviousValue9)/10;
   	P_Tem1.StanDev := SQRT(((P_Tem1.PreviousValue0 - P_Tem1.Mean10)**2 + (P_Tem1.PreviousValue1 - P_Tem1.Mean10)**2 + (P_Tem1.PreviousValue2 - P_Tem1.Mean10)**2 + (P_Tem1.PreviousValue3 - P_Tem1.Mean10)**2 + (P_Tem1.PreviousValue4 - P_Tem1.Mean10)**2 + (P_Tem1.PreviousValue5 - P_Tem1.Mean10)**2 + (P_Tem1.PreviousValue6 - P_Tem1.Mean10)**2 + (P_Tem1.PreviousValue7 - P_Tem1.Mean10)**2 + (P_Tem1.PreviousValue8 - P_Tem1.Mean10)**2 + (P_Tem1.PreviousValue9 - P_Tem1.Mean10)**2)/10);
   end_if;
END_ROUTINE

ROUTINE Update_P_Tem2   (* structured text *)
   case P_Tem2.Count of
   	0: P_Tem2.PreviousValue0 := P_Tem2.CurrentValue;
   	1: P_Tem2.PreviousValue1 := P_Tem2.CurrentValue;
   	2: P_Tem2.PreviousValue2 := P_Tem2.CurrentValue;
   	3: P_Tem2.PreviousValue3 := P_Tem2.CurrentValue;
   	4: P_Tem2.PreviousValue4 := P_Tem2.CurrentValue;
   	5: P_Tem2.PreviousValue5 := P_Tem2.CurrentValue;
   	6: P_Tem2.PreviousValue6 := P_Tem2.CurrentValue;
   	7: P_Tem2.PreviousValue7 := P_Tem2.CurrentValue;
   	8: P_Tem2.PreviousValue8 := P_Tem2.CurrentValue;
   	9: P_Tem2.PreviousValue9 := P_Tem2.CurrentValue;
   end_case;
   P_Tem2.Count := P_Tem2.Count + 1;
   if P_Tem2.Count = 10 then
   	P_Tem2.Count := 0;
   	P_Tem2.MeanStart := 1;
   end_if;
   P_Tem2.CurrentValue := Local:3:I.Ch07.Data;
   if P_Tem2.MeanStart then
   	P_Tem2.Mean10 := (P_Tem2.PreviousValue0 + P_Tem2.PreviousValue1 + P_Tem2.PreviousValue2 + P_Tem2.PreviousValue3 + P_Tem2.PreviousValue4 + P_Tem2.PreviousValue5 + P_Tem2.PreviousValue6 + P_Tem2.PreviousValue7 + P_Tem2.PreviousValue8 + P_Tem2.PreviousValue9)/10;
   	P_Tem2.StanDev := SQRT(((P_Tem2.PreviousValue0 - P_Tem2.Mean10)**2 + (P_Tem2.PreviousValue1 - P_Tem2.Mean10)**2 + (P_Tem2.PreviousValue2 - P_Tem2.Mean10)**2 + (P_Tem2.PreviousValue3 - P_Tem2.Mean10)**2 + (P_Tem2.PreviousValue4 - P_Tem2.Mean10)**2 + (P_Tem2.PreviousValue5 - P_Tem2.Mean10)**2 + (P_Tem2.PreviousValue6 - P_Tem2.Mean10)**2 + (P_Tem2.PreviousValue7 - P_Tem2.Mean10)**2 + (P_Tem2.PreviousValue8 - P_Tem2.Mean10)**2 + (P_Tem2.PreviousValue9 - P_Tem2.Mean10)**2)/10);
   end_if;
END_ROUTINE

ROUTINE Update_P_Tem3   (* structured text *)
   case P_Tem3.Count of
   	0: P_Tem3.PreviousValue0 := P_Tem3.CurrentValue;
   	1: P_Tem3.PreviousValue1 := P_Tem3.CurrentValue;
   	2: P_Tem3.PreviousValue2 := P_Tem3.CurrentValue;
   	3: P_Tem3.PreviousValue3 := P_Tem3.CurrentValue;
   	4: P_Tem3.PreviousValue4 := P_Tem3.CurrentValue;
   	5: P_Tem3.PreviousValue5 := P_Tem3.CurrentValue;
   	6: P_Tem3.PreviousValue6 := P_Tem3.CurrentValue;
   	7: P_Tem3.PreviousValue7 := P_Tem3.CurrentValue;
   	8: P_Tem3.PreviousValue8 := P_Tem3.CurrentValue;
   	9: P_Tem3.PreviousValue9 := P_Tem3.CurrentValue;
   end_case;
   P_Tem3.Count := P_Tem3.Count + 1;
   if P_Tem3.Count = 10 then
   	P_Tem3.Count := 0;
   	P_Tem3.MeanStart := 1;
   end_if;
   P_Tem3.CurrentValue := Local:2:I.Ch04.Data;
   if P_Tem3.MeanStart then
   	P_Tem3.Mean10 := (P_Tem3.PreviousValue0 + P_Tem3.PreviousValue1 + P_Tem3.PreviousValue2 + P_Tem3.PreviousValue3 + P_Tem3.PreviousValue4 + P_Tem3.PreviousValue5 + P_Tem3.PreviousValue6 + P_Tem3.PreviousValue7 + P_Tem3.PreviousValue8 + P_Tem3.PreviousValue9)/10;
   	P_Tem3.StanDev := SQRT(((P_Tem3.PreviousValue0 - P_Tem3.Mean10)**2 + (P_Tem3.PreviousValue1 - P_Tem3.Mean10)**2 + (P_Tem3.PreviousValue2 - P_Tem3.Mean10)**2 + (P_Tem3.PreviousValue3 - P_Tem3.Mean10)**2 + (P_Tem3.PreviousValue4 - P_Tem3.Mean10)**2 + (P_Tem3.PreviousValue5 - P_Tem3.Mean10)**2 + (P_Tem3.PreviousValue6 - P_Tem3.Mean10)**2 + (P_Tem3.PreviousValue7 - P_Tem3.Mean10)**2 + (P_Tem3.PreviousValue8 - P_Tem3.Mean10)**2 + (P_Tem3.PreviousValue9 - P_Tem3.Mean10)**2)/10);
   end_if;
END_ROUTINE

ROUTINE Update_P_Tem4   (* structured text *)
   case P_Tem4.Count of
   	0: P_Tem4.PreviousValue0 := P_Tem4.CurrentValue;
   	1: P_Tem4.PreviousValue1 := P_Tem4.CurrentValue;
   	2: P_Tem4.PreviousValue2 := P_Tem4.CurrentValue;
   	3: P_Tem4.PreviousValue3 := P_Tem4.CurrentValue;
   	4: P_Tem4.PreviousValue4 := P_Tem4.CurrentValue;
   	5: P_Tem4.PreviousValue5 := P_Tem4.CurrentValue;
   	6: P_Tem4.PreviousValue6 := P_Tem4.CurrentValue;
   	7: P_Tem4.PreviousValue7 := P_Tem4.CurrentValue;
   	8: P_Tem4.PreviousValue8 := P_Tem4.CurrentValue;
   	9: P_Tem4.PreviousValue9 := P_Tem4.CurrentValue;
   end_case;
   P_Tem4.Count := P_Tem4.Count + 1;
   if P_Tem4.Count = 10 then
   	P_Tem4.Count := 0;
   	P_Tem4.MeanStart := 1;
   end_if;
   P_Tem4.CurrentValue := Local:2:I.Ch05.Data;
   if P_Tem4.MeanStart then
   	P_Tem4.Mean10 := (P_Tem4.PreviousValue0 + P_Tem4.PreviousValue1 + P_Tem4.PreviousValue2 + P_Tem4.PreviousValue3 + P_Tem4.PreviousValue4 + P_Tem4.PreviousValue5 + P_Tem4.PreviousValue6 + P_Tem4.PreviousValue7 + P_Tem4.PreviousValue8 + P_Tem4.PreviousValue9)/10;
   	P_Tem4.StanDev := SQRT(((P_Tem4.PreviousValue0 - P_Tem4.Mean10)**2 + (P_Tem4.PreviousValue1 - P_Tem4.Mean10)**2 + (P_Tem4.PreviousValue2 - P_Tem4.Mean10)**2 + (P_Tem4.PreviousValue3 - P_Tem4.Mean10)**2 + (P_Tem4.PreviousValue4 - P_Tem4.Mean10)**2 + (P_Tem4.PreviousValue5 - P_Tem4.Mean10)**2 + (P_Tem4.PreviousValue6 - P_Tem4.Mean10)**2 + (P_Tem4.PreviousValue7 - P_Tem4.Mean10)**2 + (P_Tem4.PreviousValue8 - P_Tem4.Mean10)**2 + (P_Tem4.PreviousValue9 - P_Tem4.Mean10)**2)/10);
   end_if;
END_ROUTINE
END_PROGRAM

PROGRAM SafetyProgram   (* main routine MainRoutine, safety *)
VAR
   S_CD1 : BOOL;
   S_STATE : DINT;
END_VAR

ROUTINE MainRoutine   (* ladder *)
END_ROUTINE
END_PROGRAM
